LIN {X 0,Y 234.968,Z 259.216,A -85,B 0,C 180,E1 -19822.885,E2 -19822.885} C_VEL
LIN {X 0,Y 234.975,Z 259.214,A -85,B 0,C 180,E1 -19826.659,E2 -19826.659} C_VEL
LIN {X 0,Y 234.93,Z 259.221,A -85,B 0,C 180,E1 -19830.571,E2 -19830.571} C_VEL
LIN {X 0,Y 234.94,Z 259.221,A -85,B 0,C 180,E1 -19834.639,E2 -19834.639} C_VEL
LIN {X 0,Y 235.025,Z 259.387,A -85,B 0,C 180,E1 -19836.361,E2 -19836.361} C_VEL
LIN {X 0,Y 235.772,Z 263.846,A -85,B 0,C 180,E1 -19840.982,E2 -19840.982} C_VEL
LIN {X 0,Y 236.606,Z 268.443,A -85,B 0,C 180,E1 -19845.473,E2 -19845.473} C_VEL
LIN {X 0,Y 237.453,Z 272.706,A -85,B 0,C 180,E1 -19849.371,E2 -19849.371} C_VEL
LIN {X 0,Y 237.77,Z 275.178,A -85,B 0,C 180,E1 -19851.538,E2 -19851.538} C_VEL
LIN {X 0,Y 237.539,Z 276.271,A -85,B 0,C 180,E1 -19852.442,E2 -19852.442} C_VEL
LIN {X 0,Y 236.676,Z 277.419,A -85,B 0,C 180,E1 -19853.326,E2 -19853.326} C_VEL
LIN {X 0,Y 233.876,Z 279.774,A -85,B 0,C 180,E1 -19855.046,E2 -19855.046} C_VEL
LIN {X 0,Y 230.833,Z 282.181,A -85,B 0,C 180,E1 -19856.803,E2 -19856.803} C_VEL
LIN {X 0,Y 229.345,Z 283.979,A -85,B 0,C 180,E1 -19858.189,E2 -19858.189} C_VEL
LIN {X 0,Y 229.137,Z 284.57,A -85,B 0,C 180,E1 -19858.667,E2 -19858.667} C_VEL
LIN {X 0,Y 228.747,Z 286.319,A -85,B 0,C 180,E1 -19860.094,E2 -19860.094} C_VEL
LIN {X 0,Y 231.153,Z 300.125,A -85,B 0,C 180,E1 -19861.215,E2 -19861.215} C_VEL
LIN {X 0,Y 232.977,Z 313.771,A -85,B 0,C 180,E1 -19862.666,E2 -19862.666} C_VEL
LIN {X 0,Y 234.069,Z 325.973,A -85,B 0,C 180,E1 -19864.263,E2 -19864.263} C_VEL
LIN {X 0,Y 234.595,Z 337.731,A -85,B 0,C 180,E1 -19866.144,E2 -19866.144} C_VEL
LIN {X 0,Y 234.553,Z 342.841,A -85,B 0,C 180,E1 -19867.074,E2 -19867.074} C_VEL
LIN {X 0,Y 232.73,Z 351.383,A -85,B 0,C 180,E1 -19868.753,E2 -19868.753} C_VEL
LIN {X 0,Y 230.779,Z 360.913,A -85,B 0,C 180,E1 -19871.069,E2 -19871.069} C_VEL
LIN {X 0,Y 229.119,Z 368.99,A -85,B 0,C 180,E1 -19873.516,E2 -19873.516} C_VEL
LIN {X 0,Y 227.674,Z 375.926,A -85,B 0,C 180,E1 -19876.158,E2 -19876.158} C_VEL
LIN {X 0,Y 226.624,Z 382.296,A -85,B 0,C 180,E1 -19879.276,E2 -19879.276} C_VEL
LIN {X 0,Y 226.093,Z 386.448,A -85,B 0,C 180,E1 -19881.958,E2 -19881.958} C_VEL
LIN {X 0,Y 225.93,Z 389.517,A -85,B 0,C 180,E1 -19884.644,E2 -19884.644} C_VEL
LIN {X 0,Y 225.896,Z 391.02,A -85,B 0,C 180,E1 -19886.432,E2 -19886.432} C_VEL
LIN {X 0,Y 225.902,Z 392.054,A -85,B 0,C 180,E1 -19888.216,E2 -19888.216} C_VEL
LIN {X 0,Y 225.952,Z 392.675,A -85,B 0,C 180,E1 -19889.999,E2 -19889.999} C_VEL
LIN {X 0,Y 225.889,Z 392.888,A -85,B 0,C 180,E1 -19891.782,E2 -19891.782} C_VEL
LIN {X 0,Y 225.836,Z 392.705,A -85,B 0,C 180,E1 -19893.567,E2 -19893.567} C_VEL
LIN {X 0,Y 225.85,Z 392.091,A -85,B 0,C 180,E1 -19895.356,E2 -19895.356} C_VEL
LIN {X 0,Y 226.172,Z 389.669,A -85,B 0,C 180,E1 -19898.937,E2 -19898.937} C_VEL
LIN {X 0,Y 226.872,Z 386.782,A -85,B 0,C 180,E1 -19901.615,E2 -19901.615} C_VEL
LIN {X 0,Y 227.949,Z 382.909,A -85,B 0,C 180,E1 -19904.278,E2 -19904.278} C_VEL
LIN {X 0,Y 229.699,Z 377.964,A -85,B 0,C 180,E1 -19906.897,E2 -19906.897} C_VEL
LIN {X 0,Y 231.812,Z 371.807,A -85,B 0,C 180,E1 -19909.48,E2 -19909.48} C_VEL
LIN {X 0,Y 234.196,Z 364.248,A -85,B 0,C 180,E1 -19912.03,E2 -19912.03} C_VEL
LIN {X 0,Y 236.743,Z 356.653,A -85,B 0,C 180,E1 -19914.09,E2 -19914.09} C_VEL
LIN {X 0,Y 239.503,Z 347.574,A -85,B 0,C 180,E1 -19916.113,E2 -19916.113} C_VEL
LIN {X 0,Y 240.749,Z 336.486,A -85,B 0,C 180,E1 -19918.353,E2 -19918.353} C_VEL
LIN {X 0,Y 240.901,Z 325.735,A -85,B 0,C 180,E1 -19920.292,E2 -19920.292} C_VEL
LIN {X 0,Y 239.993,Z 315.116,A -85,B 0,C 180,E1 -19922.104,E2 -19922.104} C_VEL
LIN {X 0,Y 238.133,Z 304.29,A -85,B 0,C 180,E1 -19923.87,E2 -19923.87} C_VEL
LIN {X 0,Y 234.398,Z 291.005,A -85,B 0,C 180,E1 -19926.087,E2 -19926.087} C_VEL
LIN {X 0,Y 232.93,Z 286.928,A -85,B 0,C 180,E1 -19926.783,E2 -19926.783} C_VEL
LIN {X 0,Y 231.631,Z 283.737,A -85,B 0,C 180,E1 -19927.359,E2 -19927.359} C_VEL
LIN {X 0,Y 231.38,Z 282.361,A -85,B 0,C 180,E1 -19927.584,E2 -19927.584} C_VEL
LIN {X 0,Y 231.276,Z 279.496,A -85,B 0,C 180,E1 -19930.559,E2 -19930.559} C_VEL
LIN {X 0,Y 230.731,Z 276.118,A -85,B 0,C 180,E1 -19934.471,E2 -19934.471} C_VEL
LIN {X 0,Y 230.294,Z 273.504,A -85,B 0,C 180,E1 -19937.823,E2 -19937.823} C_VEL
LIN {X 0,Y 229.789,Z 270.45,A -85,B 0,C 180,E1 -19942.285,E2 -19942.285} C_VEL
LIN {X 0,Y 229.339,Z 268.039,A -85,B 0,C 180,E1 -19946.52,E2 -19946.52} C_VEL
LIN {X 0,Y 229.005,Z 266.125,A -85,B 0,C 180,E1 -19950.589,E2 -19950.589} C_VEL
LIN {X 0,Y 228.784,Z 264.663,A -85,B 0,C 180,E1 -19954.526,E2 -19954.526} C_VEL
LIN {X 0,Y 228.596,Z 263.623,A -85,B 0,C 180,E1 -19958.348,E2 -19958.348} C_VEL
LIN {X 0,Y 228.533,Z 262.899,A -85,B 0,C 180,E1 -19962.423,E2 -19962.423} C_VEL
LIN {X 0,Y 228.531,Z 262.566,A -85,B 0,C 180,E1 -19965.755,E2 -19965.755} C_VEL
LIN {X 0,Y 228.671,Z 262.482,A -85,B 0,C 180,E1 -19969.567,E2 -19969.567} C_VEL
LIN {X 0,Y 228.775,Z 262.67,A -85,B 0,C 180,E1 -19972.939,E2 -19972.939} C_VEL
LIN {X 0,Y 229.094,Z 263.408,A -85,B 0,C 180,E1 -19978.239,E2 -19978.239} C_VEL
LIN {X 0,Y 229.288,Z 263.758,A -85,B 0,C 180,E1 -19979.997,E2 -19979.997} C_VEL
LIN {X 0,Y 229.113,Z 265.292,A -85,B 0,C 180,E1 -19985.277,E2 -19985.277} C_VEL
LIN {X 0,Y 229.191,Z 266.612,A -85,B 0,C 180,E1 -19989.039,E2 -19989.039} C_VEL
LIN {X 0,Y 230.476,Z 269.741,A -85,B 0,C 180,E1 -19989.707,E2 -19989.707} C_VEL
LIN {X 0,Y 231.953,Z 271.819,A -85,B 0,C 180,E1 -19990.289,E2 -19990.289} C_VEL
LIN {X 0,Y 235.796,Z 279.227,A -85,B 0,C 180,E1 -19992.039,E2 -19992.039} C_VEL
LIN {X 0,Y 239.845,Z 288.945,A -85,B 0,C 180,E1 -19994.164,E2 -19994.164} C_VEL
LIN {X 0,Y 242.982,Z 299.405,A -85,B 0,C 180,E1 -19996.377,E2 -19996.377} C_VEL
LIN {X 0,Y 244.71,Z 309.094,A -85,B 0,C 180,E1 -19998.413,E2 -19998.413} C_VEL
LIN {X 0,Y 245.106,Z 313.998,A -85,B 0,C 180,E1 -19999.467,E2 -19999.467} C_VEL
LIN {X 0,Y 242.135,Z 324.686,A -85,B 0,C 180,E1 -20001.409,E2 -20001.409} C_VEL
LIN {X 0,Y 239.125,Z 334.171,A -85,B 0,C 180,E1 -20003.601,E2 -20003.601} C_VEL
LIN {X 0,Y 236.313,Z 342.387,A -85,B 0,C 180,E1 -20005.999,E2 -20005.999} C_VEL
LIN {X 0,Y 233.458,Z 349.872,A -85,B 0,C 180,E1 -20008.79,E2 -20008.79} C_VEL
LIN {X 0,Y 231.136,Z 355.679,A -85,B 0,C 180,E1 -20011.641,E2 -20011.641} C_VEL
LIN {X 0,Y 229.446,Z 359.674,A -85,B 0,C 180,E1 -20014.208,E2 -20014.208} C_VEL
LIN {X 0,Y 228.148,Z 362.637,A -85,B 0,C 180,E1 -20016.784,E2 -20016.784} C_VEL
LIN {X 0,Y 227.137,Z 364.655,A -85,B 0,C 180,E1 -20019.329,E2 -20019.329} C_VEL
LIN {X 0,Y 226.411,Z 365.821,A -85,B 0,C 180,E1 -20021.844,E2 -20021.844} C_VEL
LIN {X 0,Y 225.954,Z 366.155,A -85,B 0,C 180,E1 -20024.327,E2 -20024.327} C_VEL
LIN {X 0,Y 225.751,Z 365.739,A -85,B 0,C 180,E1 -20026.774,E2 -20026.774} C_VEL
LIN {X 0,Y 225.78,Z 364.618,A -85,B 0,C 180,E1 -20029.182,E2 -20029.182} C_VEL
LIN {X 0,Y 226.089,Z 362.754,A -85,B 0,C 180,E1 -20031.561,E2 -20031.561} C_VEL
LIN {X 0,Y 226.821,Z 358.635,A -85,B 0,C 180,E1 -20035.027,E2 -20035.027} C_VEL
LIN {X 0,Y 227.584,Z 354.595,A -85,B 0,C 180,E1 -20037.5,E2 -20037.5} C_VEL
LIN {X 0,Y 228.855,Z 348.086,A -85,B 0,C 180,E1 -20040.572,E2 -20040.572} C_VEL
LIN {X 0,Y 230.47,Z 340.722,A -85,B 0,C 180,E1 -20043.271,E2 -20043.271} C_VEL
LIN {X 0,Y 232.279,Z 331.67,A -85,B 0,C 180,E1 -20045.893,E2 -20045.893} C_VEL
LIN {X 0,Y 234.23,Z 322.215,A -85,B 0,C 180,E1 -20048.082,E2 -20048.082} C_VEL
LIN {X 0,Y 236.047,Z 312.051,A -85,B 0,C 180,E1 -20049.978,E2 -20049.978} C_VEL
LIN {X 0,Y 237.456,Z 303.625,A -85,B 0,C 180,E1 -20051.27,E2 -20051.27} C_VEL
LIN {X 0,Y 235.73,Z 293.055,A -85,B 0,C 180,E1 -20052.901,E2 -20052.901} C_VEL
LIN {X 0,Y 233.046,Z 281.209,A -85,B 0,C 180,E1 -20054.477,E2 -20054.477} C_VEL
LIN {X 0,Y 229.531,Z 268.807,A -85,B 0,C 180,E1 -20055.879,E2 -20055.879} C_VEL
LIN {X 0,Y 227.267,Z 261.563,A -85,B 0,C 180,E1 -20056.59,E2 -20056.59} C_VEL
LIN {X 0,Y 227.547,Z 260.142,A -85,B 0,C 180,E1 -20059.322,E2 -20059.322} C_VEL
LIN {X 0,Y 228.133,Z 260.069,A -85,B 0,C 180,E1 -20062.923,E2 -20062.923} C_VEL
LIN {X 0,Y 228.542,Z 260.018,A -85,B 0,C 180,E1 -20068.239,E2 -20068.239} C_VEL
LIN {X 0,Y 228.542,Z 260.016,A -85,B 0,C 180,E1 -20071.763,E2 -20071.763} C_VEL
LIN {X 0,Y 228.342,Z 260.04,A -85,B 0,C 180,E1 -20077.073,E2 -20077.073} C_VEL
LIN {X 0,Y 228.15,Z 260.066,A -85,B 0,C 180,E1 -20080.652,E2 -20080.652} C_VEL
LIN {X 0,Y 228.053,Z 260.079,A -85,B 0,C 180,E1 -20086.103,E2 -20086.103} C_VEL
LIN {X 0,Y 227.959,Z 260.088,A -85,B 0,C 180,E1 -20089.825,E2 -20089.825} C_VEL
LIN {X 0,Y 227.929,Z 260.094,A -85,B 0,C 180,E1 -20093.632,E2 -20093.632} C_VEL
LIN {X 0,Y 227.876,Z 260.096,A -85,B 0,C 180,E1 -20097.557,E2 -20097.557} C_VEL
LIN {X 0,Y 227.863,Z 260.101,A -85,B 0,C 180,E1 -20101.624,E2 -20101.624} C_VEL
LIN {X 0,Y 227.892,Z 260.09,A -85,B 0,C 180,E1 -20105.871,E2 -20105.871} C_VEL
LIN {X 0,Y 227.896,Z 260.097,A -85,B 0,C 180,E1 -20110.363,E2 -20110.363} C_VEL
LIN {X 0,Y 227.913,Z 260.091,A -85,B 0,C 180,E1 -20114.832,E2 -20114.832} C_VEL
LIN {X 0,Y 227.928,Z 260.081,A -85,B 0,C 180,E1 -20117.735,E2 -20117.735} C_VEL
LIN {X 0,Y 227.875,Z 260.098,A -85,B 0,C 180,E1 -20121.92,E2 -20121.92} C_VEL
LIN {X 0,Y 227.886,Z 260.096,A -85,B 0,C 180,E1 -20126.376,E2 -20126.376} C_VEL
LIN {X 0,Y 227.915,Z 260.085,A -85,B 0,C 180,E1 -20130.441,E2 -20130.441} C_VEL
LIN {X 0,Y 227.926,Z 260.093,A -85,B 0,C 180,E1 -20134.429,E2 -20134.429} C_VEL
LIN {X 0,Y 227.961,Z 260.087,A -85,B 0,C 180,E1 -20138.29,E2 -20138.29} C_VEL
LIN {X 0,Y 228.035,Z 260.067,A -85,B 0,C 180,E1 -20142.829,E2 -20142.829} C_VEL
LIN {X 0,Y 228.073,Z 260.073,A -85,B 0,C 180,E1 -20147.546,E2 -20147.546} C_VEL
LIN {X 0,Y 228.265,Z 260.049,A -85,B 0,C 180,E1 -20151.148,E2 -20151.148} C_VEL
LIN {X 0,Y 228.32,Z 260.038,A -85,B 0,C 180,E1 -20152.931,E2 -20152.931} C_VEL
LIN {X 0,Y 228.557,Z 260.012,A -85,B 0,C 180,E1 -20158.241,E2 -20158.241} C_VEL
LIN {X 0,Y 228.556,Z 260.017,A -85,B 0,C 180,E1 -20161.765,E2 -20161.765} C_VEL
LIN {X 0,Y 228.315,Z 260.035,A -85,B 0,C 180,E1 -20167.076,E2 -20167.076} C_VEL
LIN {X 0,Y 228.15,Z 260.063,A -85,B 0,C 180,E1 -20170.654,E2 -20170.654} C_VEL
LIN {X 0,Y 228.068,Z 260.072,A -85,B 0,C 180,E1 -20174.275,E2 -20174.275} C_VEL
LIN {X 0,Y 228.01,Z 260.081,A -85,B 0,C 180,E1 -20177.956,E2 -20177.956} C_VEL
LIN {X 0,Y 227.938,Z 260.091,A -85,B 0,C 180,E1 -20182.331,E2 -20182.331} C_VEL
LIN {X 0,Y 227.95,Z 260.09,A -85,B 0,C 180,E1 -20186.604,E2 -20186.604} C_VEL
LIN {X 0,Y 227.905,Z 260.095,A -85,B 0,C 180,E1 -20190.293,E2 -20190.293} C_VEL
LIN {X 0,Y 227.941,Z 260.093,A -85,B 0,C 180,E1 -20195.66,E2 -20195.66} C_VEL
LIN {X 0,Y 228.549,Z 263.853,A -85,B 0,C 180,E1 -20199.756,E2 -20199.756} C_VEL
LIN {X 0,Y 229.234,Z 267.624,A -85,B 0,C 180,E1 -20203.618,E2 -20203.618} C_VEL
LIN {X 0,Y 230.1,Z 271.927,A -85,B 0,C 180,E1 -20207.781,E2 -20207.781} C_VEL
LIN {X 0,Y 230.71,Z 275.958,A -85,B 0,C 180,E1 -20211.467,E2 -20211.467} C_VEL
LIN {X 0,Y 230.34,Z 279.576,A -85,B 0,C 180,E1 -20214.568,E2 -20214.568} C_VEL
LIN {X 0,Y 229.137,Z 284.57,A -85,B 0,C 180,E1 -20218.667,E2 -20218.667} C_VEL
LIN {X 0,Y 228.886,Z 286.269,A -85,B 0,C 180,E1 -20219.369,E2 -20219.369} C_VEL
LIN {X 0,Y 228.442,Z 289.896,A -85,B 0,C 180,E1 -20220.027,E2 -20220.027} C_VEL
LIN {X 0,Y 227.746,Z 295.552,A -85,B 0,C 180,E1 -20220.531,E2 -20220.531} C_VEL
LIN {X 0,Y 226.19,Z 306.821,A -85,B 0,C 180,E1 -20221.327,E2 -20221.327} C_VEL
LIN {X 0,Y 226.038,Z 313.153,A -85,B 0,C 180,E1 -20221.971,E2 -20221.971} C_VEL
LIN {X 0,Y 227.096,Z 325.04,A -85,B 0,C 180,E1 -20223.563,E2 -20223.563} C_VEL
LIN {X 0,Y 227.636,Z 336.145,A -85,B 0,C 180,E1 -20225.367,E2 -20225.367} C_VEL
LIN {X 0,Y 227.471,Z 343.759,A -85,B 0,C 180,E1 -20226.8,E2 -20226.8} C_VEL
LIN {X 0,Y 225.655,Z 352.086,A -85,B 0,C 180,E1 -20228.533,E2 -20228.533} C_VEL
LIN {X 0,Y 223.699,Z 361.369,A -85,B 0,C 180,E1 -20230.906,E2 -20230.906} C_VEL
LIN {X 0,Y 222.002,Z 369.289,A -85,B 0,C 180,E1 -20233.445,E2 -20233.445} C_VEL
LIN {X 0,Y 220.535,Z 376.088,A -85,B 0,C 180,E1 -20236.171,E2 -20236.171} C_VEL
LIN {X 0,Y 219.619,Z 381.53,A -85,B 0,C 180,E1 -20238.929,E2 -20238.929} C_VEL
LIN {X 0,Y 219.055,Z 385.761,A -85,B 0,C 180,E1 -20241.698,E2 -20241.698} C_VEL
LIN {X 0,Y 218.895,Z 388.906,A -85,B 0,C 180,E1 -20244.472,E2 -20244.472} C_VEL
LIN {X 0,Y 218.818,Z 390.443,A -85,B 0,C 180,E1 -20246.316,E2 -20246.316} C_VEL
LIN {X 0,Y 218.834,Z 391.542,A -85,B 0,C 180,E1 -20248.159,E2 -20248.159} C_VEL
LIN {X 0,Y 218.88,Z 392.194,A -85,B 0,C 180,E1 -20249.999,E2 -20249.999} C_VEL
LIN {X 0,Y 218.819,Z 392.439,A -85,B 0,C 180,E1 -20251.84,E2 -20251.84} C_VEL
LIN {X 0,Y 218.774,Z 391.862,A -85,B 0,C 180,E1 -20255.192,E2 -20255.192} C_VEL
LIN {X 0,Y 218.862,Z 390.765,A -85,B 0,C 180,E1 -20257.379,E2 -20257.379} C_VEL
LIN {X 0,Y 219.595,Z 387.639,A -85,B 0,C 180,E1 -20261.07,E2 -20261.07} C_VEL
LIN {X 0,Y 220.583,Z 384.174,A -85,B 0,C 180,E1 -20263.824,E2 -20263.824} C_VEL
LIN {X 0,Y 222.242,Z 379.682,A -85,B 0,C 180,E1 -20266.534,E2 -20266.534} C_VEL
LIN {X 0,Y 224.7,Z 373.034,A -85,B 0,C 180,E1 -20269.646,E2 -20269.646} C_VEL
LIN {X 0,Y 227.17,Z 365.861,A -85,B 0,C 180,E1 -20272.269,E2 -20272.269} C_VEL
LIN {X 0,Y 230.312,Z 357.056,A -85,B 0,C 180,E1 -20274.807,E2 -20274.807} C_VEL
LIN {X 0,Y 232.709,Z 350.054,A -85,B 0,C 180,E1 -20276.452,E2 -20276.452} C_VEL
LIN {X 0,Y 234.258,Z 339.819,A -85,B 0,C 180,E1 -20278.685,E2 -20278.685} C_VEL
LIN {X 0,Y 234.848,Z 330.187,A -85,B 0,C 180,E1 -20280.579,E2 -20280.579} C_VEL
LIN {X 0,Y 234.313,Z 318.822,A -85,B 0,C 180,E1 -20282.675,E2 -20282.675} C_VEL
LIN {X 0,Y 232.75,Z 307.621,A -85,B 0,C 180,E1 -20284.644,E2 -20284.644} C_VEL
LIN {X 0,Y 229.499,Z 294.855,A -85,B 0,C 180,E1 -20286.943,E2 -20286.943} C_VEL
LIN {X 0,Y 227.903,Z 290.354,A -85,B 0,C 180,E1 -20287.808,E2 -20287.808} C_VEL
LIN {X 0,Y 226.657,Z 286.91,A -85,B 0,C 180,E1 -20288.466,E2 -20288.466} C_VEL
LIN {X 0,Y 224.857,Z 283.567,A -85,B 0,C 180,E1 -20289.282,E2 -20289.282} C_VEL
LIN {X 0,Y 224.416,Z 281.713,A -85,B 0,C 180,E1 -20289.576,E2 -20289.576} C_VEL
LIN {X 0,Y 223.899,Z 278.116,A -85,B 0,C 180,E1 -20293.781,E2 -20293.781} C_VEL
LIN {X 0,Y 223.242,Z 274.481,A -85,B 0,C 180,E1 -20298.612,E2 -20298.612} C_VEL
LIN {X 0,Y 222.783,Z 271.534,A -85,B 0,C 180,E1 -20303.171,E2 -20303.171} C_VEL
LIN {X 0,Y 222.31,Z 269.239,A -85,B 0,C 180,E1 -20307.488,E2 -20307.488} C_VEL
LIN {X 0,Y 222.047,Z 267.418,A -85,B 0,C 180,E1 -20311.653,E2 -20311.653} C_VEL
LIN {X 0,Y 221.826,Z 266.071,A -85,B 0,C 180,E1 -20315.675,E2 -20315.675} C_VEL
LIN {X 0,Y 221.662,Z 265.125,A -85,B 0,C 180,E1 -20319.585,E2 -20319.585} C_VEL
LIN {X 0,Y 221.643,Z 264.523,A -85,B 0,C 180,E1 -20323.416,E2 -20323.416} C_VEL
LIN {X 0,Y 221.619,Z 264.242,A -85,B 0,C 180,E1 -20327.171,E2 -20327.171} C_VEL
LIN {X 0,Y 221.845,Z 264.216,A -85,B 0,C 180,E1 -20330.883,E2 -20330.883} C_VEL
LIN {X 0,Y 221.832,Z 264.527,A -85,B 0,C 180,E1 -20334.543,E2 -20334.543} C_VEL
LIN {X 0,Y 222.176,Z 265.025,A -85,B 0,C 180,E1 -20338.184,E2 -20338.184} C_VEL
LIN {X 0,Y 222.363,Z 265.346,A -85,B 0,C 180,E1 -20339.997,E2 -20339.997} C_VEL
LIN {X 0,Y 222.164,Z 266.305,A -85,B 0,C 180,E1 -20343.624,E2 -20343.624} C_VEL
LIN {X 0,Y 222.271,Z 267.329,A -85,B 0,C 180,E1 -20346.978,E2 -20346.978} C_VEL
LIN {X 0,Y 223.527,Z 270.421,A -85,B 0,C 180,E1 -20347.676,E2 -20347.676} C_VEL
LIN {X 0,Y 225.456,Z 272.865,A -85,B 0,C 180,E1 -20348.512,E2 -20348.512} C_VEL
LIN {X 0,Y 227.344,Z 276.202,A -85,B 0,C 180,E1 -20349.441,E2 -20349.441} C_VEL
LIN {X 0,Y 231.257,Z 284.148,A -85,B 0,C 180,E1 -20351.45,E2 -20351.45} C_VEL
LIN {X 0,Y 235.059,Z 294.303,A -85,B 0,C 180,E1 -20353.836,E2 -20353.836} C_VEL
LIN {X 0,Y 237.429,Z 303.385,A -85,B 0,C 180,E1 -20355.888,E2 -20355.888} C_VEL
LIN {X 0,Y 238.808,Z 312.702,A -85,B 0,C 180,E1 -20357.996,E2 -20357.996} C_VEL
LIN {X 0,Y 239.049,Z 315.526,A -85,B 0,C 180,E1 -20358.653,E2 -20358.653} C_VEL
LIN {X 0,Y 236.225,Z 325.137,A -85,B 0,C 180,E1 -20360.458,E2 -20360.458} C_VEL
LIN {X 0,Y 233.007,Z 334.695,A -85,B 0,C 180,E1 -20362.722,E2 -20362.722} C_VEL
LIN {X 0,Y 229.837,Z 343.388,A -85,B 0,C 180,E1 -20365.343,E2 -20365.343} C_VEL
LIN {X 0,Y 227.401,Z 349.398,A -85,B 0,C 180,E1 -20367.615,E2 -20367.615} C_VEL
LIN {X 0,Y 225.313,Z 354.324,A -85,B 0,C 180,E1 -20369.935,E2 -20369.935} C_VEL
LIN {X 0,Y 223.53,Z 358.337,A -85,B 0,C 180,E1 -20372.306,E2 -20372.306} C_VEL
LIN {X 0,Y 222.035,Z 361.528,A -85,B 0,C 180,E1 -20374.728,E2 -20374.728} C_VEL
LIN {X 0,Y 220.827,Z 364.005,A -85,B 0,C 180,E1 -20377.286,E2 -20377.286} C_VEL
LIN {X 0,Y 219.863,Z 365.671,A -85,B 0,C 180,E1 -20379.902,E2 -20379.902} C_VEL
LIN {X 0,Y 219.183,Z 366.482,A -85,B 0,C 180,E1 -20382.484,E2 -20382.484} C_VEL
LIN {X 0,Y 218.774,Z 366.526,A -85,B 0,C 180,E1 -20385.031,E2 -20385.031} C_VEL
LIN {X 0,Y 218.664,Z 365.782,A -85,B 0,C 180,E1 -20387.661,E2 -20387.661} C_VEL
LIN {X 0,Y 218.819,Z 364.114,A -85,B 0,C 180,E1 -20390.422,E2 -20390.422} C_VEL
LIN {X 0,Y 219.503,Z 360.447,A -85,B 0,C 180,E1 -20394.044,E2 -20394.044} C_VEL
LIN {X 0,Y 220.338,Z 355.883,A -85,B 0,C 180,E1 -20397.165,E2 -20397.165} C_VEL
LIN {X 0,Y 221.506,Z 350.33,A -85,B 0,C 180,E1 -20400.02,E2 -20400.02} C_VEL
LIN {X 0,Y 223.152,Z 342.814,A -85,B 0,C 180,E1 -20403.018,E2 -20403.018} C_VEL
LIN {X 0,Y 224.873,Z 334.614,A -85,B 0,C 180,E1 -20405.616,E2 -20405.616} C_VEL
LIN {X 0,Y 226.786,Z 325.461,A -85,B 0,C 180,E1 -20407.931,E2 -20407.931} C_VEL
LIN {X 0,Y 228.794,Z 315.178,A -85,B 0,C 180,E1 -20410.019,E2 -20410.019} C_VEL
LIN {X 0,Y 230.676,Z 304.573,A -85,B 0,C 180,E1 -20411.746,E2 -20411.746} C_VEL
LIN {X 0,Y 228.759,Z 293.176,A -85,B 0,C 180,E1 -20413.58,E2 -20413.58} C_VEL
LIN {X 0,Y 226.135,Z 281.8,A -85,B 0,C 180,E1 -20415.145,E2 -20415.145} C_VEL
LIN {X 0,Y 222.615,Z 269.482,A -85,B 0,C 180,E1 -20416.595,E2 -20416.595} C_VEL
LIN {X 0,Y 220.286,Z 261.958,A -85,B 0,C 180,E1 -20417.389,E2 -20417.389} C_VEL
LIN {X 0,Y 220.423,Z 261.03,A -85,B 0,C 180,E1 -20418.972,E2 -20418.972} C_VEL
LIN {X 0,Y 220.843,Z 260.976,A -85,B 0,C 180,E1 -20420.845,E2 -20420.845} C_VEL
LIN {X 0,Y 221.053,Z 260.95,A -85,B 0,C 180,E1 -20422.695,E2 -20422.695} C_VEL
LIN {X 0,Y 221.499,Z 260.895,A -85,B 0,C 180,E1 -20428.183,E2 -20428.183} C_VEL
LIN {X 0,Y 221.5,Z 260.893,A -85,B 0,C 180,E1 -20431.819,E2 -20431.819} C_VEL
LIN {X 0,Y 221.277,Z 260.921,A -85,B 0,C 180,E1 -20437.3,E2 -20437.3} C_VEL
LIN {X 0,Y 221.099,Z 260.944,A -85,B 0,C 180,E1 -20440.996,E2 -20440.996} C_VEL
LIN {X 0,Y 221.013,Z 260.958,A -85,B 0,C 180,E1 -20446.631,E2 -20446.631} C_VEL
LIN {X 0,Y 220.914,Z 260.967,A -85,B 0,C 180,E1 -20450.485,E2 -20450.485} C_VEL
LIN {X 0,Y 220.872,Z 260.975,A -85,B 0,C 180,E1 -20454.435,E2 -20454.435} C_VEL
LIN {X 0,Y 220.827,Z 260.976,A -85,B 0,C 180,E1 -20458.516,E2 -20458.516} C_VEL
LIN {X 0,Y 220.814,Z 260.981,A -85,B 0,C 180,E1 -20462.757,E2 -20462.757} C_VEL
LIN {X 0,Y 220.829,Z 260.971,A -85,B 0,C 180,E1 -20467.291,E2 -20467.291} C_VEL
LIN {X 0,Y 220.866,Z 260.972,A -85,B 0,C 180,E1 -20471.931,E2 -20471.931} C_VEL
LIN {X 0,Y 220.868,Z 260.966,A -85,B 0,C 180,E1 -20475.575,E2 -20475.575} C_VEL
LIN {X 0,Y 220.855,Z 260.968,A -85,B 0,C 180,E1 -20479.795,E2 -20479.795} C_VEL
LIN {X 0,Y 220.834,Z 260.977,A -85,B 0,C 180,E1 -20482.799,E2 -20482.799} C_VEL
LIN {X 0,Y 220.821,Z 260.972,A -85,B 0,C 180,E1 -20487.249,E2 -20487.249} C_VEL
LIN {X 0,Y 220.833,Z 260.967,A -85,B 0,C 180,E1 -20491.49,E2 -20491.49} C_VEL
LIN {X 0,Y 220.865,Z 260.971,A -85,B 0,C 180,E1 -20495.569,E2 -20495.569} C_VEL
LIN {X 0,Y 220.892,Z 260.966,A -85,B 0,C 180,E1 -20499.517,E2 -20499.517} C_VEL
LIN {X 0,Y 221.017,Z 260.941,A -85,B 0,C 180,E1 -20503.374,E2 -20503.374} C_VEL
LIN {X 0,Y 221.013,Z 260.951,A -85,B 0,C 180,E1 -20507.142,E2 -20507.142} C_VEL
LIN {X 0,Y 221.203,Z 260.928,A -85,B 0,C 180,E1 -20510.863,E2 -20510.863} C_VEL
LIN {X 0,Y 221.138,Z 260.928,A -85,B 0,C 180,E1 -20514.532,E2 -20514.532} C_VEL
LIN {X 0,Y 221.515,Z 260.89,A -85,B 0,C 180,E1 -20518.185,E2 -20518.185} C_VEL
LIN {X 0,Y 221.514,Z 260.893,A -85,B 0,C 180,E1 -20521.821,E2 -20521.821} C_VEL
LIN {X 0,Y 221.252,Z 260.915,A -85,B 0,C 180,E1 -20527.303,E2 -20527.303} C_VEL
LIN {X 0,Y 221.072,Z 260.946,A -85,B 0,C 180,E1 -20530.999,E2 -20530.999} C_VEL
LIN {X 0,Y 221.023,Z 260.945,A -85,B 0,C 180,E1 -20536.632,E2 -20536.632} C_VEL
LIN {X 0,Y 220.9,Z 260.967,A -85,B 0,C 180,E1 -20540.488,E2 -20540.488} C_VEL
LIN {X 0,Y 220.875,Z 260.971,A -85,B 0,C 180,E1 -20544.437,E2 -20544.437} C_VEL
LIN {X 0,Y 220.835,Z 260.976,A -85,B 0,C 180,E1 -20548.517,E2 -20548.517} C_VEL
LIN {X 0,Y 220.825,Z 260.979,A -85,B 0,C 180,E1 -20552.758,E2 -20552.758} C_VEL
LIN {X 0,Y 220.877,Z 260.996,A -85,B 0,C 180,E1 -20555.223,E2 -20555.223} C_VEL
LIN {X 0,Y 221.254,Z 262.925,A -85,B 0,C 180,E1 -20557.427,E2 -20557.427} C_VEL
LIN {X 0,Y 221.897,Z 266.859,A -85,B 0,C 180,E1 -20561.695,E2 -20561.695} C_VEL
LIN {X 0,Y 222.786,Z 271.605,A -85,B 0,C 180,E1 -20566.519,E2 -20566.519} C_VEL
LIN {X 0,Y 223.477,Z 275.311,A -85,B 0,C 180,E1 -20570.071,E2 -20570.071} C_VEL
LIN {X 0,Y 223.647,Z 277.167,A -85,B 0,C 180,E1 -20571.781,E2 -20571.781} C_VEL
LIN {X 0,Y 223.513,Z 278.882,A -85,B 0,C 180,E1 -20573.313,E2 -20573.313} C_VEL
LIN {X 0,Y 222.349,Z 283.787,A -85,B 0,C 180,E1 -20577.497,E2 -20577.497} C_VEL
LIN {X 0,Y 221.883,Z 285.968,A -85,B 0,C 180,E1 -20579.337,E2 -20579.337} C_VEL
LIN {X 0,Y 224.328,Z 300.095,A -85,B 0,C 180,E1 -20580.542,E2 -20580.542} C_VEL
LIN {X 0,Y 226.038,Z 313.153,A -85,B 0,C 180,E1 -20581.971,E2 -20581.971} C_VEL
LIN {X 0,Y 225.877,Z 318.574,A -85,B 0,C 180,E1 -20582.594,E2 -20582.594} C_VEL
LIN {X 0,Y 223.763,Z 327.332,A -85,B 0,C 180,E1 -20583.633,E2 -20583.633} C_VEL
LIN {X 0,Y 221.358,Z 335.781,A -85,B 0,C 180,E1 -20584.842,E2 -20584.842} C_VEL
LIN {X 0,Y 220.763,Z 340.626,A -85,B 0,C 180,E1 -20585.721,E2 -20585.721} C_VEL
LIN {X 0,Y 220.379,Z 344.579,A -85,B 0,C 180,E1 -20586.506,E2 -20586.506} C_VEL
LIN {X 0,Y 218.232,Z 354.538,A -85,B 0,C 180,E1 -20588.758,E2 -20588.758} C_VEL
LIN {X 0,Y 216.456,Z 362.736,A -85,B 0,C 180,E1 -20591.053,E2 -20591.053} C_VEL
LIN {X 0,Y 214.634,Z 370.768,A -85,B 0,C 180,E1 -20593.839,E2 -20593.839} C_VEL
LIN {X 0,Y 213.19,Z 377.204,A -85,B 0,C 180,E1 -20596.657,E2 -20596.657} C_VEL
LIN {X 0,Y 212.38,Z 382.317,A -85,B 0,C 180,E1 -20599.513,E2 -20599.513} C_VEL
LIN {X 0,Y 211.879,Z 386.252,A -85,B 0,C 180,E1 -20602.375,E2 -20602.375} C_VEL
LIN {X 0,Y 211.801,Z 388.524,A -85,B 0,C 180,E1 -20604.565,E2 -20604.565} C_VEL
LIN {X 0,Y 211.767,Z 391.002,A -85,B 0,C 180,E1 -20608.097,E2 -20608.097} C_VEL
LIN {X 0,Y 211.81,Z 391.706,A -85,B 0,C 180,E1 -20609.999,E2 -20609.999} C_VEL
LIN {X 0,Y 211.75,Z 391.988,A -85,B 0,C 180,E1 -20611.901,E2 -20611.901} C_VEL
LIN {X 0,Y 211.692,Z 391.56,A -85,B 0,C 180,E1 -20615.116,E2 -20615.116} C_VEL
LIN {X 0,Y 211.795,Z 390.459,A -85,B 0,C 180,E1 -20617.626,E2 -20617.626} C_VEL
LIN {X 0,Y 212.579,Z 387.408,A -85,B 0,C 180,E1 -20621.44,E2 -20621.44} C_VEL
LIN {X 0,Y 213.673,Z 384.042,A -85,B 0,C 180,E1 -20624.28,E2 -20624.28} C_VEL
LIN {X 0,Y 215.433,Z 379.663,A -85,B 0,C 180,E1 -20627.073,E2 -20627.073} C_VEL
LIN {X 0,Y 217.583,Z 374.159,A -85,B 0,C 180,E1 -20629.824,E2 -20629.824} C_VEL
LIN {X 0,Y 220.148,Z 367.371,A -85,B 0,C 180,E1 -20632.524,E2 -20632.524} C_VEL
LIN {X 0,Y 223.297,Z 359.059,A -85,B 0,C 180,E1 -20635.143,E2 -20635.143} C_VEL
LIN {X 0,Y 226.353,Z 350.665,A -85,B 0,C 180,E1 -20637.255,E2 -20637.255} C_VEL
LIN {X 0,Y 228.08,Z 340.743,A -85,B 0,C 180,E1 -20639.538,E2 -20639.538} C_VEL
LIN {X 0,Y 228.786,Z 331.404,A -85,B 0,C 180,E1 -20641.48,E2 -20641.48} C_VEL
LIN {X 0,Y 228.371,Z 319.541,A -85,B 0,C 180,E1 -20643.804,E2 -20643.804} C_VEL
LIN {X 0,Y 226.908,Z 308.652,A -85,B 0,C 180,E1 -20645.878,E2 -20645.878} C_VEL
LIN {X 0,Y 223.933,Z 296.118,A -85,B 0,C 180,E1 -20648.312,E2 -20648.312} C_VEL
LIN {X 0,Y 222.113,Z 291.312,A -85,B 0,C 180,E1 -20649.379,E2 -20649.379} C_VEL
LIN {X 0,Y 220.479,Z 287.639,A -85,B 0,C 180,E1 -20650.258,E2 -20650.258} C_VEL
LIN {X 0,Y 219.61,Z 286.184,A -85,B 0,C 180,E1 -20650.672,E2 -20650.672} C_VEL
LIN {X 0,Y 217.643,Z 282.698,A -85,B 0,C 180,E1 -20651.675,E2 -20651.675} C_VEL
LIN {X 0,Y 217.155,Z 280.93,A -85,B 0,C 180,E1 -20652.041,E2 -20652.041} C_VEL
LIN {X 0,Y 216.636,Z 278.198,A -85,B 0,C 180,E1 -20655.536,E2 -20655.536} C_VEL
LIN {X 0,Y 216.221,Z 275.45,A -85,B 0,C 180,E1 -20659.449,E2 -20659.449} C_VEL
LIN {X 0,Y 215.749,Z 272.652,A -85,B 0,C 180,E1 -20664.099,E2 -20664.099} C_VEL
LIN {X 0,Y 215.391,Z 270.436,A -85,B 0,C 180,E1 -20668.526,E2 -20668.526} C_VEL
LIN {X 0,Y 215.106,Z 268.732,A -85,B 0,C 180,E1 -20672.777,E2 -20672.777} C_VEL
LIN {X 0,Y 214.913,Z 267.482,A -85,B 0,C 180,E1 -20676.892,E2 -20676.892} C_VEL
LIN {X 0,Y 214.774,Z 266.51,A -85,B 0,C 180,E1 -20681.611,E2 -20681.611} C_VEL
LIN {X 0,Y 214.75,Z 266.124,A -85,B 0,C 180,E1 -20684.819,E2 -20684.819} C_VEL
LIN {X 0,Y 214.949,Z 265.918,A -85,B 0,C 180,E1 -20690.588,E2 -20690.588} C_VEL
LIN {X 0,Y 214.951,Z 266.188,A -85,B 0,C 180,E1 -20694.368,E2 -20694.368} C_VEL
LIN {X 0,Y 215.263,Z 266.652,A -85,B 0,C 180,E1 -20698.126,E2 -20698.126} C_VEL
LIN {X 0,Y 215.464,Z 266.952,A -85,B 0,C 180,E1 -20699.997,E2 -20699.997} C_VEL
LIN {X 0,Y 215.284,Z 268.304,A -85,B 0,C 180,E1 -20704.561,E2 -20704.561} C_VEL
LIN {X 0,Y 216.369,Z 270.889,A -85,B 0,C 180,E1 -20705.238,E2 -20705.238} C_VEL
LIN {X 0,Y 218.727,Z 273.665,A -85,B 0,C 180,E1 -20706.397,E2 -20706.397} C_VEL
LIN {X 0,Y 220.5,Z 276.89,A -85,B 0,C 180,E1 -20707.379,E2 -20707.379} C_VEL
LIN {X 0,Y 221.503,Z 278.267,A -85,B 0,C 180,E1 -20707.868,E2 -20707.868} C_VEL
LIN {X 0,Y 226.408,Z 288.487,A -85,B 0,C 180,E1 -20710.731,E2 -20710.731} C_VEL
LIN {X 0,Y 229.337,Z 296.745,A -85,B 0,C 180,E1 -20712.834,E2 -20712.834} C_VEL
LIN {X 0,Y 231.579,Z 305.929,A -85,B 0,C 180,E1 -20715.064,E2 -20715.064} C_VEL
LIN {X 0,Y 232.713,Z 314.419,A -85,B 0,C 180,E1 -20717.121,E2 -20717.121} C_VEL
LIN {X 0,Y 232.766,Z 317.983,A -85,B 0,C 180,E1 -20717.971,E2 -20717.971} C_VEL
LIN {X 0,Y 229.348,Z 328.691,A -85,B 0,C 180,E1 -20720.149,E2 -20720.149} C_VEL
LIN {X 0,Y 226.163,Z 337.372,A -85,B 0,C 180,E1 -20722.371,E2 -20722.371} C_VEL
LIN {X 0,Y 223.309,Z 344.619,A -85,B 0,C 180,E1 -20724.715,E2 -20724.715} C_VEL
LIN {X 0,Y 220.819,Z 350.343,A -85,B 0,C 180,E1 -20726.984,E2 -20726.984} C_VEL
LIN {X 0,Y 217.857,Z 356.813,A -85,B 0,C 180,E1 -20730.331,E2 -20730.331} C_VEL
LIN {X 0,Y 215.545,Z 361.513,A -85,B 0,C 180,E1 -20733.658,E2 -20733.658} C_VEL
LIN {X 0,Y 214.221,Z 364.019,A -85,B 0,C 180,E1 -20736.19,E2 -20736.19} C_VEL
LIN {X 0,Y 213.128,Z 365.787,A -85,B 0,C 180,E1 -20738.79,E2 -20738.79} C_VEL
LIN {X 0,Y 212.323,Z 366.808,A -85,B 0,C 180,E1 -20741.448,E2 -20741.448} C_VEL
LIN {X 0,Y 211.781,Z 367.054,A -85,B 0,C 180,E1 -20744.173,E2 -20744.173} C_VEL
LIN {X 0,Y 211.565,Z 366.439,A -85,B 0,C 180,E1 -20746.949,E2 -20746.949} C_VEL
LIN {X 0,Y 211.651,Z 364.927,A -85,B 0,C 180,E1 -20749.788,E2 -20749.788} C_VEL
LIN {X 0,Y 212.251,Z 361.648,A -85,B 0,C 180,E1 -20753.417,E2 -20753.417} C_VEL
LIN {X 0,Y 212.83,Z 358.535,A -85,B 0,C 180,E1 -20755.851,E2 -20755.851} C_VEL
LIN {X 0,Y 213.806,Z 353.805,A -85,B 0,C 180,E1 -20758.713,E2 -20758.713} C_VEL
LIN {X 0,Y 215.275,Z 347.156,A -85,B 0,C 180,E1 -20761.81,E2 -20761.81} C_VEL
LIN {X 0,Y 216.923,Z 339.75,A -85,B 0,C 180,E1 -20764.538,E2 -20764.538} C_VEL
LIN {X 0,Y 218.827,Z 331.157,A -85,B 0,C 180,E1 -20767.083,E2 -20767.083} C_VEL
LIN {X 0,Y 221.021,Z 320.731,A -85,B 0,C 180,E1 -20769.527,E2 -20769.527} C_VEL
LIN {X 0,Y 223.274,Z 309.248,A -85,B 0,C 180,E1 -20771.654,E2 -20771.654} C_VEL
LIN {X 0,Y 223.85,Z 305.239,A -85,B 0,C 180,E1 -20772.29,E2 -20772.29} C_VEL
LIN {X 0,Y 221.934,Z 294.164,A -85,B 0,C 180,E1 -20774.151,E2 -20774.151} C_VEL
LIN {X 0,Y 219.228,Z 282.313,A -85,B 0,C 180,E1 -20775.852,E2 -20775.852} C_VEL
LIN {X 0,Y 215.583,Z 269.746,A -85,B 0,C 180,E1 -20777.408,E2 -20777.408} C_VEL
LIN {X 0,Y 213.3,Z 262.4,A -85,B 0,C 180,E1 -20778.177,E2 -20778.177} C_VEL
LIN {X 0,Y 213.705,Z 261.865,A -85,B 0,C 180,E1 -20780.584,E2 -20780.584} C_VEL
LIN {X 0,Y 213.977,Z 261.832,A -85,B 0,C 180,E1 -20782.452,E2 -20782.452} C_VEL
LIN {X 0,Y 214.431,Z 261.776,A -85,B 0,C 180,E1 -20788.123,E2 -20788.123} C_VEL
LIN {X 0,Y 214.541,Z 261.762,A -85,B 0,C 180,E1 -20790.001,E2 -20790.001} C_VEL
LIN {X 0,Y 214.433,Z 261.773,A -85,B 0,C 180,E1 -20791.879,E2 -20791.879} C_VEL
LIN {X 0,Y 214.215,Z 261.801,A -85,B 0,C 180,E1 -20797.542,E2 -20797.542} C_VEL
LIN {X 0,Y 214.032,Z 261.821,A -85,B 0,C 180,E1 -20801.364,E2 -20801.364} C_VEL
LIN {X 0,Y 213.926,Z 261.841,A -85,B 0,C 180,E1 -20805.238,E2 -20805.238} C_VEL
LIN {X 0,Y 213.873,Z 261.843,A -85,B 0,C 180,E1 -20809.185,E2 -20809.185} C_VEL
LIN {X 0,Y 213.852,Z 261.85,A -85,B 0,C 180,E1 -20813.227,E2 -20813.227} C_VEL
LIN {X 0,Y 213.818,Z 261.847,A -85,B 0,C 180,E1 -20817.452,E2 -20817.452} C_VEL
LIN {X 0,Y 213.77,Z 261.857,A -85,B 0,C 180,E1 -20821.738,E2 -20821.738} C_VEL
LIN {X 0,Y 213.745,Z 261.852,A -85,B 0,C 180,E1 -20826.289,E2 -20826.289} C_VEL
LIN {X 0,Y 213.817,Z 261.851,A -85,B 0,C 180,E1 -20831.102,E2 -20831.102} C_VEL
LIN {X 0,Y 213.829,Z 261.847,A -85,B 0,C 180,E1 -20833.696,E2 -20833.696} C_VEL
LIN {X 0,Y 213.834,Z 261.84,A -85,B 0,C 180,E1 -20836.359,E2 -20836.359} C_VEL
LIN {X 0,Y 213.818,Z 261.844,A -85,B 0,C 180,E1 -20839.113,E2 -20839.113} C_VEL
LIN {X 0,Y 213.752,Z 261.858,A -85,B 0,C 180,E1 -20843.718,E2 -20843.718} C_VEL
LIN {X 0,Y 213.792,Z 261.842,A -85,B 0,C 180,E1 -20848.728,E2 -20848.728} C_VEL
LIN {X 0,Y 213.823,Z 261.846,A -85,B 0,C 180,E1 -20852.607,E2 -20852.607} C_VEL
LIN {X 0,Y 213.851,Z 261.845,A -85,B 0,C 180,E1 -20856.956,E2 -20856.956} C_VEL
LIN {X 0,Y 213.944,Z 261.821,A -85,B 0,C 180,E1 -20862.807,E2 -20862.807} C_VEL
LIN {X 0,Y 213.954,Z 261.831,A -85,B 0,C 180,E1 -20866.71,E2 -20866.71} C_VEL
LIN {X 0,Y 214.141,Z 261.808,A -85,B 0,C 180,E1 -20870.559,E2 -20870.559} C_VEL
LIN {X 0,Y 214.099,Z 261.804,A -85,B 0,C 180,E1 -20874.352,E2 -20874.352} C_VEL
LIN {X 0,Y 214.448,Z 261.77,A -85,B 0,C 180,E1 -20878.125,E2 -20878.125} C_VEL
LIN {X 0,Y 214.554,Z 261.76,A -85,B 0,C 180,E1 -20880.003,E2 -20880.003} C_VEL
LIN {X 0,Y 214.447,Z 261.773,A -85,B 0,C 180,E1 -20881.881,E2 -20881.881} C_VEL
LIN {X 0,Y 214.192,Z 261.795,A -85,B 0,C 180,E1 -20887.545,E2 -20887.545} C_VEL
LIN {X 0,Y 214.004,Z 261.828,A -85,B 0,C 180,E1 -20891.367,E2 -20891.367} C_VEL
LIN {X 0,Y 213.939,Z 261.832,A -85,B 0,C 180,E1 -20895.24,E2 -20895.24} C_VEL
LIN {X 0,Y 213.847,Z 261.846,A -85,B 0,C 180,E1 -20899.19,E2 -20899.19} C_VEL
LIN {X 0,Y 213.855,Z 261.848,A -85,B 0,C 180,E1 -20903.229,E2 -20903.229} C_VEL
LIN {X 0,Y 213.837,Z 261.85,A -85,B 0,C 180,E1 -20907.452,E2 -20907.452} C_VEL
LIN {X 0,Y 213.776,Z 261.857,A -85,B 0,C 180,E1 -20911.739,E2 -20911.739} C_VEL
LIN {X 0,Y 213.83,Z 261.9,A -85,B 0,C 180,E1 -20914.745,E2 -20914.745} C_VEL
LIN {X 0,Y 214.553,Z 266.176,A -85,B 0,C 180,E1 -20919.702,E2 -20919.702} C_VEL
LIN {X 0,Y 215.281,Z 270.243,A -85,B 0,C 180,E1 -20924.092,E2 -20924.092} C_VEL
LIN {X 0,Y 216.159,Z 274.484,A -85,B 0,C 180,E1 -20928.404,E2 -20928.404} C_VEL
LIN {X 0,Y 216.559,Z 278.132,A -85,B 0,C 180,E1 -20931.93,E2 -20931.93} C_VEL
LIN {X 0,Y 216.144,Z 280.841,A -85,B 0,C 180,E1 -20934.383,E2 -20934.383} C_VEL
LIN {X 0,Y 214.99,Z 285.553,A -85,B 0,C 180,E1 -20938.526,E2 -20938.526} C_VEL
LIN {X 0,Y 217.464,Z 299.872,A -85,B 0,C 180,E1 -20939.805,E2 -20939.805} C_VEL
LIN {X 0,Y 219.251,Z 313.785,A -85,B 0,C 180,E1 -20941.404,E2 -20941.404} C_VEL
LIN {X 0,Y 220.248,Z 325.451,A -85,B 0,C 180,E1 -20943.05,E2 -20943.05} C_VEL
LIN {X 0,Y 220.734,Z 337.109,A -85,B 0,C 180,E1 -20945.046,E2 -20945.046} C_VEL
LIN {X 0,Y 220.763,Z 340.626,A -85,B 0,C 180,E1 -20945.721,E2 -20945.721} C_VEL
LIN {X 0,Y 219.896,Z 343.77,A -85,B 0,C 180,E1 -20946.305,E2 -20946.305} C_VEL
LIN {X 0,Y 217.9,Z 346.692,A -85,B 0,C 180,E1 -20946.814,E2 -20946.814} C_VEL
LIN {X 0,Y 212.337,Z 352.998,A -85,B 0,C 180,E1 -20948.027,E2 -20948.027} C_VEL
LIN {X 0,Y 210.992,Z 355.788,A -85,B 0,C 180,E1 -20948.726,E2 -20948.726} C_VEL
LIN {X 0,Y 209.01,Z 364.532,A -85,B 0,C 180,E1 -20951.37,E2 -20951.37} C_VEL
LIN {X 0,Y 207.261,Z 372.093,A -85,B 0,C 180,E1 -20954.259,E2 -20954.259} C_VEL
LIN {X 0,Y 205.902,Z 378.161,A -85,B 0,C 180,E1 -20957.181,E2 -20957.181} C_VEL
LIN {X 0,Y 205.147,Z 382.969,A -85,B 0,C 180,E1 -20960.136,E2 -20960.136} C_VEL
LIN {X 0,Y 204.749,Z 386.627,A -85,B 0,C 180,E1 -20963.099,E2 -20963.099} C_VEL
LIN {X 0,Y 204.675,Z 389.239,A -85,B 0,C 180,E1 -20966.061,E2 -20966.061} C_VEL
LIN {X 0,Y 204.702,Z 390.439,A -85,B 0,C 180,E1 -20968.031,E2 -20968.031} C_VEL
LIN {X 0,Y 204.741,Z 391.216,A -85,B 0,C 180,E1 -20969.999,E2 -20969.999} C_VEL
LIN {X 0,Y 204.68,Z 391.537,A -85,B 0,C 180,E1 -20971.967,E2 -20971.967} C_VEL
LIN {X 0,Y 204.586,Z 390.993,A -85,B 0,C 180,E1 -20975.914,E2 -20975.914} C_VEL
LIN {X 0,Y 204.721,Z 390.147,A -85,B 0,C 180,E1 -20977.892,E2 -20977.892} C_VEL
LIN {X 0,Y 205.068,Z 388.879,A -85,B 0,C 180,E1 -20979.866,E2 -20979.866} C_VEL
LIN {X 0,Y 206.279,Z 385.132,A -85,B 0,C 180,E1 -20983.796,E2 -20983.796} C_VEL
LIN {X 0,Y 207.96,Z 381.191,A -85,B 0,C 180,E1 -20986.693,E2 -20986.693} C_VEL
LIN {X 0,Y 210.045,Z 376.177,A -85,B 0,C 180,E1 -20989.547,E2 -20989.547} C_VEL
LIN {X 0,Y 212.824,Z 369.641,A -85,B 0,C 180,E1 -20992.473,E2 -20992.473} C_VEL
LIN {X 0,Y 215.738,Z 362.408,A -85,B 0,C 180,E1 -20995.054,E2 -20995.054} C_VEL
LIN {X 0,Y 219.497,Z 353.038,A -85,B 0,C 180,E1 -20997.662,E2 -20997.662} C_VEL
LIN {X 0,Y 221.395,Z 344.717,A -85,B 0,C 180,E1 -20999.735,E2 -20999.735} C_VEL
LIN {X 0,Y 222.612,Z 334.953,A -85,B 0,C 180,E1 -21001.93,E2 -21001.93} C_VEL
LIN {X 0,Y 222.719,Z 324.229,A -85,B 0,C 180,E1 -21004.215,E2 -21004.215} C_VEL
LIN {X 0,Y 221.754,Z 313.166,A -85,B 0,C 180,E1 -21006.464,E2 -21006.464} C_VEL
LIN {X 0,Y 219.653,Z 302.214,A -85,B 0,C 180,E1 -21008.757,E2 -21008.757} C_VEL
LIN {X 0,Y 217.631,Z 295.876,A -85,B 0,C 180,E1 -21010.229,E2 -21010.229} C_VEL
LIN {X 0,Y 215.729,Z 291.477,A -85,B 0,C 180,E1 -21011.411,E2 -21011.411} C_VEL
LIN {X 0,Y 213.703,Z 287.405,A -85,B 0,C 180,E1 -21012.615,E2 -21012.615} C_VEL
LIN {X 0,Y 213.027,Z 286.115,A -85,B 0,C 180,E1 -21013.004,E2 -21013.004} C_VEL
LIN {X 0,Y 210.695,Z 282.747,A -85,B 0,C 180,E1 -21014.284,E2 -21014.284} C_VEL
LIN {X 0,Y 209.762,Z 280.047,A -85,B 0,C 180,E1 -21015,E2 -21015} C_VEL
LIN {X 0,Y 209.428,Z 278.076,A -85,B 0,C 180,E1 -21017.84,E2 -21017.84} C_VEL
LIN {X 0,Y 209.171,Z 276.298,A -85,B 0,C 180,E1 -21020.602,E2 -21020.602} C_VEL
LIN {X 0,Y 208.733,Z 273.791,A -85,B 0,C 180,E1 -21025.08,E2 -21025.08} C_VEL
LIN {X 0,Y 208.372,Z 271.688,A -85,B 0,C 180,E1 -21029.604,E2 -21029.604} C_VEL
LIN {X 0,Y 208.118,Z 270.087,A -85,B 0,C 180,E1 -21033.957,E2 -21033.957} C_VEL
LIN {X 0,Y 207.949,Z 268.937,A -85,B 0,C 180,E1 -21038.172,E2 -21038.172} C_VEL
LIN {X 0,Y 207.884,Z 268.177,A -85,B 0,C 180,E1 -21042.283,E2 -21042.283} C_VEL
LIN {X 0,Y 207.858,Z 267.764,A -85,B 0,C 180,E1 -21046.306,E2 -21046.306} C_VEL
LIN {X 0,Y 208.047,Z 267.63,A -85,B 0,C 180,E1 -21050.273,E2 -21050.273} C_VEL
LIN {X 0,Y 208.054,Z 267.847,A -85,B 0,C 180,E1 -21054.181,E2 -21054.181} C_VEL
LIN {X 0,Y 208.562,Z 268.582,A -85,B 0,C 180,E1 -21059.997,E2 -21059.997} C_VEL
LIN {X 0,Y 208.496,Z 269.066,A -85,B 0,C 180,E1 -21061.747,E2 -21061.747} C_VEL
LIN {X 0,Y 209.511,Z 271.7,A -85,B 0,C 180,E1 -21062.521,E2 -21062.521} C_VEL
LIN {X 0,Y 211.944,Z 274.534,A -85,B 0,C 180,E1 -21063.918,E2 -21063.918} C_VEL
LIN {X 0,Y 213.867,Z 277.921,A -85,B 0,C 180,E1 -21065.123,E2 -21065.123} C_VEL
LIN {X 0,Y 214.85,Z 278.932,A -85,B 0,C 180,E1 -21065.628,E2 -21065.628} C_VEL
LIN {X 0,Y 219.078,Z 287.047,A -85,B 0,C 180,E1 -21068.297,E2 -21068.297} C_VEL
LIN {X 0,Y 222.12,Z 294.503,A -85,B 0,C 180,E1 -21070.47,E2 -21070.47} C_VEL
LIN {X 0,Y 224.552,Z 302.58,A -85,B 0,C 180,E1 -21072.652,E2 -21072.652} C_VEL
LIN {X 0,Y 226.187,Z 311.15,A -85,B 0,C 180,E1 -21074.896,E2 -21074.896} C_VEL
LIN {X 0,Y 226.792,Z 317.975,A -85,B 0,C 180,E1 -21076.654,E2 -21076.654} C_VEL
LIN {X 0,Y 226.764,Z 319.791,A -85,B 0,C 180,E1 -21077.12,E2 -21077.12} C_VEL
LIN {X 0,Y 223.328,Z 329.855,A -85,B 0,C 180,E1 -21079.255,E2 -21079.255} C_VEL
LIN {X 0,Y 219.811,Z 338.717,A -85,B 0,C 180,E1 -21081.638,E2 -21081.638} C_VEL
LIN {X 0,Y 216.231,Z 347.013,A -85,B 0,C 180,E1 -21084.489,E2 -21084.489} C_VEL
LIN {X 0,Y 213.096,Z 353.721,A -85,B 0,C 180,E1 -21087.494,E2 -21087.494} C_VEL
LIN {X 0,Y 210.966,Z 358.033,A -85,B 0,C 180,E1 -21089.989,E2 -21089.989} C_VEL
LIN {X 0,Y 208.948,Z 361.752,A -85,B 0,C 180,E1 -21092.769,E2 -21092.769} C_VEL
LIN {X 0,Y 207.382,Z 364.479,A -85,B 0,C 180,E1 -21095.579,E2 -21095.579} C_VEL
LIN {X 0,Y 206.172,Z 366.301,A -85,B 0,C 180,E1 -21098.372,E2 -21098.372} C_VEL
LIN {X 0,Y 205.302,Z 367.288,A -85,B 0,C 180,E1 -21101.141,E2 -21101.141} C_VEL
LIN {X 0,Y 204.735,Z 367.501,A -85,B 0,C 180,E1 -21103.875,E2 -21103.875} C_VEL
LIN {X 0,Y 204.515,Z 366.921,A -85,B 0,C 180,E1 -21106.586,E2 -21106.586} C_VEL
LIN {X 0,Y 204.514,Z 365.626,A -85,B 0,C 180,E1 -21109.239,E2 -21109.239} C_VEL
LIN {X 0,Y 204.857,Z 363.412,A -85,B 0,C 180,E1 -21112.091,E2 -21112.091} C_VEL
LIN {X 0,Y 205.545,Z 360.02,A -85,B 0,C 180,E1 -21115.139,E2 -21115.139} C_VEL
LIN {X 0,Y 206.518,Z 355.275,A -85,B 0,C 180,E1 -21118.288,E2 -21118.288} C_VEL
LIN {X 0,Y 207.91,Z 348.965,A -85,B 0,C 180,E1 -21121.499,E2 -21121.499} C_VEL
LIN {X 0,Y 209.492,Z 342.37,A -85,B 0,C 180,E1 -21124.145,E2 -21124.145} C_VEL
LIN {X 0,Y 211.364,Z 333.967,A -85,B 0,C 180,E1 -21126.855,E2 -21126.855} C_VEL
LIN {X 0,Y 213.502,Z 324.594,A -85,B 0,C 180,E1 -21129.277,E2 -21129.277} C_VEL
LIN {X 0,Y 215.692,Z 313.989,A -85,B 0,C 180,E1 -21131.478,E2 -21131.478} C_VEL
LIN {X 0,Y 216.987,Z 306.19,A -85,B 0,C 180,E1 -21132.811,E2 -21132.811} C_VEL
LIN {X 0,Y 215.033,Z 294.581,A -85,B 0,C 180,E1 -21134.844,E2 -21134.844} C_VEL
LIN {X 0,Y 212.345,Z 282.831,A -85,B 0,C 180,E1 -21136.605,E2 -21136.605} C_VEL
LIN {X 0,Y 208.537,Z 269.817,A -85,B 0,C 180,E1 -21138.273,E2 -21138.273} C_VEL
LIN {X 0,Y 206.345,Z 262.799,A -85,B 0,C 180,E1 -21139.069,E2 -21139.069} C_VEL
LIN {X 0,Y 206.892,Z 262.715,A -85,B 0,C 180,E1 -21142.192,E2 -21142.192} C_VEL
LIN {X 0,Y 207.367,Z 262.657,A -85,B 0,C 180,E1 -21148.059,E2 -21148.059} C_VEL
LIN {X 0,Y 207.505,Z 262.639,A -85,B 0,C 180,E1 -21150.001,E2 -21150.001} C_VEL
LIN {X 0,Y 207.074,Z 262.69,A -85,B 0,C 180,E1 -21153.893,E2 -21153.893} C_VEL
LIN {X 0,Y 207.155,Z 262.68,A -85,B 0,C 180,E1 -21157.8,E2 -21157.8} C_VEL
LIN {X 0,Y 206.969,Z 262.699,A -85,B 0,C 180,E1 -21161.757,E2 -21161.757} C_VEL
LIN {X 0,Y 206.865,Z 262.719,A -85,B 0,C 180,E1 -21165.772,E2 -21165.772} C_VEL
LIN {X 0,Y 206.812,Z 262.723,A -85,B 0,C 180,E1 -21169.867,E2 -21169.867} C_VEL
LIN {X 0,Y 206.762,Z 262.731,A -85,B 0,C 180,E1 -21174.073,E2 -21174.073} C_VEL
LIN {X 0,Y 206.734,Z 262.73,A -85,B 0,C 180,E1 -21178.421,E2 -21178.421} C_VEL
LIN {X 0,Y 206.7,Z 262.738,A -85,B 0,C 180,E1 -21182.959,E2 -21182.959} C_VEL
LIN {X 0,Y 206.717,Z 262.728,A -85,B 0,C 180,E1 -21187.733,E2 -21187.733} C_VEL
LIN {X 0,Y 206.742,Z 262.731,A -85,B 0,C 180,E1 -21191.6,E2 -21191.6} C_VEL
LIN {X 0,Y 206.739,Z 262.725,A -85,B 0,C 180,E1 -21195.553,E2 -21195.553} C_VEL
LIN {X 0,Y 206.738,Z 262.726,A -85,B 0,C 180,E1 -21199.772,E2 -21199.772} C_VEL
LIN {X 0,Y 206.727,Z 262.733,A -85,B 0,C 180,E1 -21204.699,E2 -21204.699} C_VEL
LIN {X 0,Y 206.72,Z 262.721,A -85,B 0,C 180,E1 -21209.343,E2 -21209.343} C_VEL
LIN {X 0,Y 206.73,Z 262.73,A -85,B 0,C 180,E1 -21213.776,E2 -21213.776} C_VEL
LIN {X 0,Y 206.757,Z 262.73,A -85,B 0,C 180,E1 -21218.047,E2 -21218.047} C_VEL
LIN {X 0,Y 206.873,Z 262.702,A -85,B 0,C 180,E1 -21222.2,E2 -21222.2} C_VEL
LIN {X 0,Y 206.896,Z 262.711,A -85,B 0,C 180,E1 -21226.248,E2 -21226.248} C_VEL
LIN {X 0,Y 207.101,Z 262.687,A -85,B 0,C 180,E1 -21230.234,E2 -21230.234} C_VEL
LIN {X 0,Y 207.06,Z 262.681,A -85,B 0,C 180,E1 -21234.159,E2 -21234.159} C_VEL
LIN {X 0,Y 207.384,Z 262.649,A -85,B 0,C 180,E1 -21238.061,E2 -21238.061} C_VEL
LIN {X 0,Y 207.518,Z 262.636,A -85,B 0,C 180,E1 -21240.003,E2 -21240.003} C_VEL
LIN {X 0,Y 207.383,Z 262.653,A -85,B 0,C 180,E1 -21241.945,E2 -21241.945} C_VEL
LIN {X 0,Y 207.136,Z 262.675,A -85,B 0,C 180,E1 -21247.803,E2 -21247.803} C_VEL
LIN {X 0,Y 206.929,Z 262.71,A -85,B 0,C 180,E1 -21251.761,E2 -21251.761} C_VEL
LIN {X 0,Y 206.873,Z 262.709,A -85,B 0,C 180,E1 -21255.773,E2 -21255.773} C_VEL
LIN {X 0,Y 206.791,Z 262.726,A -85,B 0,C 180,E1 -21259.871,E2 -21259.871} C_VEL
LIN {X 0,Y 206.771,Z 262.728,A -85,B 0,C 180,E1 -21264.074,E2 -21264.074} C_VEL
LIN {X 0,Y 206.745,Z 262.731,A -85,B 0,C 180,E1 -21268.422,E2 -21268.422} C_VEL
LIN {X 0,Y 206.719,Z 262.736,A -85,B 0,C 180,E1 -21272.957,E2 -21272.957} C_VEL
LIN {X 0,Y 206.8,Z 262.902,A -85,B 0,C 180,E1 -21274.405,E2 -21274.405} C_VEL
LIN {X 0,Y 207.403,Z 266.55,A -85,B 0,C 180,E1 -21278.795,E2 -21278.795} C_VEL
LIN {X 0,Y 208.21,Z 270.934,A -85,B 0,C 180,E1 -21283.699,E2 -21283.699} C_VEL
LIN {X 0,Y 208.966,Z 274.721,A -85,B 0,C 180,E1 -21287.727,E2 -21287.727} C_VEL
LIN {X 0,Y 209.508,Z 278.69,A -85,B 0,C 180,E1 -21291.709,E2 -21291.709} C_VEL
LIN {X 0,Y 209.215,Z 280.84,A -85,B 0,C 180,E1 -21293.732,E2 -21293.732} C_VEL
LIN {X 0,Y 208.104,Z 285.186,A -85,B 0,C 180,E1 -21297.696,E2 -21297.696} C_VEL
LIN {X 0,Y 210.568,Z 299.183,A -85,B 0,C 180,E1 -21298.977,E2 -21298.977} C_VEL
LIN {X 0,Y 212.164,Z 311.41,A -85,B 0,C 180,E1 -21300.408,E2 -21300.408} C_VEL
LIN {X 0,Y 213.324,Z 324.356,A -85,B 0,C 180,E1 -21302.271,E2 -21302.271} C_VEL
LIN {X 0,Y 213.77,Z 335.569,A -85,B 0,C 180,E1 -21304.221,E2 -21304.221} C_VEL
LIN {X 0,Y 213.798,Z 343.034,A -85,B 0,C 180,E1 -21305.737,E2 -21305.737} C_VEL
LIN {X 0,Y 211.56,Z 353.252,A -85,B 0,C 180,E1 -21308.054,E2 -21308.054} C_VEL
LIN {X 0,Y 210.992,Z 355.788,A -85,B 0,C 180,E1 -21308.726,E2 -21308.726} C_VEL
LIN {X 0,Y 209.444,Z 359.808,A -85,B 0,C 180,E1 -21309.829,E2 -21309.829} C_VEL
LIN {X 0,Y 205.173,Z 365.795,A -85,B 0,C 180,E1 -21311.673,E2 -21311.673} C_VEL
LIN {X 0,Y 200.995,Z 371.161,A -85,B 0,C 180,E1 -21313.724,E2 -21313.724} C_VEL
LIN {X 0,Y 199.628,Z 374.21,A -85,B 0,C 180,E1 -21315.126,E2 -21315.126} C_VEL
LIN {X 0,Y 198.363,Z 380.706,A -85,B 0,C 180,E1 -21318.762,E2 -21318.762} C_VEL
LIN {X 0,Y 197.781,Z 384.819,A -85,B 0,C 180,E1 -21321.827,E2 -21321.827} C_VEL
LIN {X 0,Y 197.64,Z 387.676,A -85,B 0,C 180,E1 -21324.693,E2 -21324.693} C_VEL
LIN {X 0,Y 197.637,Z 389.868,A -85,B 0,C 180,E1 -21327.961,E2 -21327.961} C_VEL
LIN {X 0,Y 197.674,Z 390.695,A -85,B 0,C 180,E1 -21329.999,E2 -21329.999} C_VEL
LIN {X 0,Y 197.611,Z 391.083,A -85,B 0,C 180,E1 -21332.037,E2 -21332.037} C_VEL
LIN {X 0,Y 197.509,Z 390.621,A -85,B 0,C 180,E1 -21336.127,E2 -21336.127} C_VEL
LIN {X 0,Y 198.035,Z 388.629,A -85,B 0,C 180,E1 -21340.22,E2 -21340.22} C_VEL
LIN {X 0,Y 199.354,Z 384.976,A -85,B 0,C 180,E1 -21344.286,E2 -21344.286} C_VEL
LIN {X 0,Y 201.145,Z 381.144,A -85,B 0,C 180,E1 -21347.276,E2 -21347.276} C_VEL
LIN {X 0,Y 203.361,Z 376.264,A -85,B 0,C 180,E1 -21350.217,E2 -21350.217} C_VEL
LIN {X 0,Y 206.154,Z 370.122,A -85,B 0,C 180,E1 -21353.12,E2 -21353.12} C_VEL
LIN {X 0,Y 209.333,Z 362.772,A -85,B 0,C 180,E1 -21355.876,E2 -21355.876} C_VEL
LIN {X 0,Y 213.245,Z 353.647,A -85,B 0,C 180,E1 -21358.546,E2 -21358.546} C_VEL
LIN {X 0,Y 215.473,Z 344.594,A -85,B 0,C 180,E1 -21360.91,E2 -21360.91} C_VEL
LIN {X 0,Y 216.724,Z 335.105,A -85,B 0,C 180,E1 -21363.167,E2 -21363.167} C_VEL
LIN {X 0,Y 216.901,Z 323.888,A -85,B 0,C 180,E1 -21365.677,E2 -21365.677} C_VEL
LIN {X 0,Y 216.068,Z 313.697,A -85,B 0,C 180,E1 -21367.926,E2 -21367.926} C_VEL
LIN {X 0,Y 214.255,Z 303.979,A -85,B 0,C 180,E1 -21370.139,E2 -21370.139} C_VEL
LIN {X 0,Y 212.191,Z 297.718,A -85,B 0,C 180,E1 -21371.816,E2 -21371.816} C_VEL
LIN {X 0,Y 209.694,Z 292.179,A -85,B 0,C 180,E1 -21373.531,E2 -21373.531} C_VEL
LIN {X 0,Y 207.162,Z 287.987,A -85,B 0,C 180,E1 -21375.166,E2 -21375.166} C_VEL
LIN {X 0,Y 206.282,Z 285.759,A -85,B 0,C 180,E1 -21375.839,E2 -21375.839} C_VEL
LIN {X 0,Y 203.781,Z 282.661,A -85,B 0,C 180,E1 -21377.409,E2 -21377.409} C_VEL
LIN {X 0,Y 202.367,Z 279.024,A -85,B 0,C 180,E1 -21378.708,E2 -21378.708} C_VEL
LIN {X 0,Y 202.02,Z 276.434,A -85,B 0,C 180,E1 -21383.141,E2 -21383.141} C_VEL
LIN {X 0,Y 201.545,Z 273.872,A -85,B 0,C 180,E1 -21388.459,E2 -21388.459} C_VEL
LIN {X 0,Y 201.281,Z 272.15,A -85,B 0,C 180,E1 -21393.002,E2 -21393.002} C_VEL
LIN {X 0,Y 201.097,Z 270.892,A -85,B 0,C 180,E1 -21397.388,E2 -21397.388} C_VEL
LIN {X 0,Y 201.011,Z 270.027,A -85,B 0,C 180,E1 -21401.656,E2 -21401.656} C_VEL
LIN {X 0,Y 200.95,Z 269.546,A -85,B 0,C 180,E1 -21405.826,E2 -21405.826} C_VEL
LIN {X 0,Y 201.134,Z 269.352,A -85,B 0,C 180,E1 -21409.935,E2 -21409.935} C_VEL
LIN {X 0,Y 201.175,Z 269.512,A -85,B 0,C 180,E1 -21413.981,E2 -21413.981} C_VEL
LIN {X 0,Y 201.488,Z 270.064,A -85,B 0,C 180,E1 -21418.185,E2 -21418.185} C_VEL
LIN {X 0,Y 202.552,Z 272.403,A -85,B 0,C 180,E1 -21419.127,E2 -21419.127} C_VEL
LIN {X 0,Y 205.503,Z 275.634,A -85,B 0,C 180,E1 -21421.148,E2 -21421.148} C_VEL
LIN {X 0,Y 207.176,Z 278.802,A -85,B 0,C 180,E1 -21422.427,E2 -21422.427} C_VEL
LIN {X 0,Y 208.871,Z 281.257,A -85,B 0,C 180,E1 -21423.567,E2 -21423.567} C_VEL
LIN {X 0,Y 210.965,Z 284.463,A -85,B 0,C 180,E1 -21424.954,E2 -21424.954} C_VEL
LIN {X 0,Y 214.497,Z 291.637,A -85,B 0,C 180,E1 -21427.528,E2 -21427.528} C_VEL
LIN {X 0,Y 217.171,Z 298.774,A -85,B 0,C 180,E1 -21429.758,E2 -21429.758} C_VEL
LIN {X 0,Y 219.55,Z 308.16,A -85,B 0,C 180,E1 -21432.475,E2 -21432.475} C_VEL
LIN {X 0,Y 220.625,Z 316.354,A -85,B 0,C 180,E1 -21434.761,E2 -21434.761} C_VEL
LIN {X 0,Y 220.777,Z 321.666,A -85,B 0,C 180,E1 -21436.233,E2 -21436.233} C_VEL
LIN {X 0,Y 217.218,Z 331.342,A -85,B 0,C 180,E1 -21438.385,E2 -21438.385} C_VEL
LIN {X 0,Y 213.729,Z 339.663,A -85,B 0,C 180,E1 -21440.712,E2 -21440.712} C_VEL
LIN {X 0,Y 209.887,Z 347.995,A -85,B 0,C 180,E1 -21443.688,E2 -21443.688} C_VEL
LIN {X 0,Y 206.533,Z 354.593,A -85,B 0,C 180,E1 -21446.802,E2 -21446.802} C_VEL
LIN {X 0,Y 203.532,Z 360.149,A -85,B 0,C 180,E1 -21450.319,E2 -21450.319} C_VEL
LIN {X 0,Y 201.543,Z 363.443,A -85,B 0,C 180,E1 -21453.188,E2 -21453.188} C_VEL
LIN {X 0,Y 199.721,Z 366.215,A -85,B 0,C 180,E1 -21456.737,E2 -21456.737} C_VEL
LIN {X 0,Y 198.679,Z 367.452,A -85,B 0,C 180,E1 -21459.543,E2 -21459.543} C_VEL
LIN {X 0,Y 197.898,Z 367.948,A -85,B 0,C 180,E1 -21462.43,E2 -21462.43} C_VEL
LIN {X 0,Y 197.472,Z 367.645,A -85,B 0,C 180,E1 -21465.375,E2 -21465.375} C_VEL
LIN {X 0,Y 197.382,Z 366.477,A -85,B 0,C 180,E1 -21468.388,E2 -21468.388} C_VEL
LIN {X 0,Y 197.654,Z 364.357,A -85,B 0,C 180,E1 -21471.461,E2 -21471.461} C_VEL
LIN {X 0,Y 198.324,Z 361.188,A -85,B 0,C 180,E1 -21474.585,E2 -21474.585} C_VEL
LIN {X 0,Y 199.303,Z 356.315,A -85,B 0,C 180,E1 -21478.067,E2 -21478.067} C_VEL
LIN {X 0,Y 200.823,Z 349.696,A -85,B 0,C 180,E1 -21481.615,E2 -21481.615} C_VEL
LIN {X 0,Y 202.513,Z 342.914,A -85,B 0,C 180,E1 -21484.453,E2 -21484.453} C_VEL
LIN {X 0,Y 204.436,Z 334.564,A -85,B 0,C 180,E1 -21487.25,E2 -21487.25} C_VEL
LIN {X 0,Y 206.759,Z 324.734,A -85,B 0,C 180,E1 -21489.871,E2 -21489.871} C_VEL
LIN {X 0,Y 208.82,Z 315.063,A -85,B 0,C 180,E1 -21491.947,E2 -21491.947} C_VEL
LIN {X 0,Y 210.211,Z 307.777,A -85,B 0,C 180,E1 -21493.241,E2 -21493.241} C_VEL
LIN {X 0,Y 208.522,Z 297.042,A -85,B 0,C 180,E1 -21495.219,E2 -21495.219} C_VEL
LIN {X 0,Y 206.194,Z 286.288,A -85,B 0,C 180,E1 -21496.951,E2 -21496.951} C_VEL
LIN {X 0,Y 202.674,Z 273.565,A -85,B 0,C 180,E1 -21498.725,E2 -21498.725} C_VEL
LIN {X 0,Y 199.464,Z 263.652,A -85,B 0,C 180,E1 -21499.921,E2 -21499.921} C_VEL
LIN {X 0,Y 199.807,Z 263.598,A -85,B 0,C 180,E1 -21501.913,E2 -21501.913} C_VEL
LIN {X 0,Y 200.305,Z 263.537,A -85,B 0,C 180,E1 -21507.99,E2 -21507.99} C_VEL
LIN {X 0,Y 200.469,Z 263.515,A -85,B 0,C 180,E1 -21510.001,E2 -21510.001} C_VEL
LIN {X 0,Y 200.02,Z 263.569,A -85,B 0,C 180,E1 -21514.031,E2 -21514.031} C_VEL
LIN {X 0,Y 200.099,Z 263.559,A -85,B 0,C 180,E1 -21518.077,E2 -21518.077} C_VEL
LIN {X 0,Y 199.902,Z 263.579,A -85,B 0,C 180,E1 -21522.179,E2 -21522.179} C_VEL
LIN {X 0,Y 199.803,Z 263.599,A -85,B 0,C 180,E1 -21526.345,E2 -21526.345} C_VEL
LIN {X 0,Y 199.741,Z 263.605,A -85,B 0,C 180,E1 -21530.602,E2 -21530.602} C_VEL
LIN {X 0,Y 199.668,Z 263.613,A -85,B 0,C 180,E1 -21534.986,E2 -21534.986} C_VEL
LIN {X 0,Y 199.665,Z 263.614,A -85,B 0,C 180,E1 -21539.525,E2 -21539.525} C_VEL
LIN {X 0,Y 199.655,Z 263.617,A -85,B 0,C 180,E1 -21542.355,E2 -21542.355} C_VEL
LIN {X 0,Y 199.645,Z 263.607,A -85,B 0,C 180,E1 -21546.76,E2 -21546.76} C_VEL
LIN {X 0,Y 199.694,Z 263.608,A -85,B 0,C 180,E1 -21549.309,E2 -21549.309} C_VEL
LIN {X 0,Y 199.693,Z 263.611,A -85,B 0,C 180,E1 -21552.353,E2 -21552.353} C_VEL
LIN {X 0,Y 199.687,Z 263.604,A -85,B 0,C 180,E1 -21555.265,E2 -21555.265} C_VEL
LIN {X 0,Y 199.687,Z 263.597,A -85,B 0,C 180,E1 -21558.038,E2 -21558.038} C_VEL
LIN {X 0,Y 199.697,Z 263.608,A -85,B 0,C 180,E1 -21560.739,E2 -21560.739} C_VEL
LIN {X 0,Y 199.631,Z 263.616,A -85,B 0,C 180,E1 -21565.722,E2 -21565.722} C_VEL
LIN {X 0,Y 199.7,Z 263.6,A -85,B 0,C 180,E1 -21568.141,E2 -21568.141} C_VEL
LIN {X 0,Y 199.685,Z 263.607,A -85,B 0,C 180,E1 -21572.776,E2 -21572.776} C_VEL
LIN {X 0,Y 199.737,Z 263.603,A -85,B 0,C 180,E1 -21577.233,E2 -21577.233} C_VEL
LIN {X 0,Y 199.796,Z 263.585,A -85,B 0,C 180,E1 -21581.761,E2 -21581.761} C_VEL
LIN {X 0,Y 199.837,Z 263.586,A -85,B 0,C 180,E1 -21585.752,E2 -21585.752} C_VEL
LIN {X 0,Y 200.024,Z 263.57,A -85,B 0,C 180,E1 -21589.885,E2 -21589.885} C_VEL
LIN {X 0,Y 200.022,Z 263.559,A -85,B 0,C 180,E1 -21593.953,E2 -21593.953} C_VEL
LIN {X 0,Y 200.324,Z 263.527,A -85,B 0,C 180,E1 -21597.993,E2 -21597.993} C_VEL
LIN {X 0,Y 200.483,Z 263.512,A -85,B 0,C 180,E1 -21600.003,E2 -21600.003} C_VEL
LIN {X 0,Y 200.024,Z 263.565,A -85,B 0,C 180,E1 -21604.033,E2 -21604.033} C_VEL
LIN {X 0,Y 200.084,Z 263.556,A -85,B 0,C 180,E1 -21608.08,E2 -21608.08} C_VEL
LIN {X 0,Y 199.879,Z 263.586,A -85,B 0,C 180,E1 -21612.182,E2 -21612.182} C_VEL
LIN {X 0,Y 199.811,Z 263.587,A -85,B 0,C 180,E1 -21616.346,E2 -21616.346} C_VEL
LIN {X 0,Y 199.708,Z 263.607,A -85,B 0,C 180,E1 -21620.608,E2 -21620.608} C_VEL
LIN {X 0,Y 199.681,Z 263.612,A -85,B 0,C 180,E1 -21624.987,E2 -21624.987} C_VEL
LIN {X 0,Y 199.673,Z 263.614,A -85,B 0,C 180,E1 -21629.526,E2 -21629.526} C_VEL
LIN {X 0,Y 199.717,Z 263.671,A -85,B 0,C 180,E1 -21633.738,E2 -21633.738} C_VEL
LIN {X 0,Y 200.272,Z 266.972,A -85,B 0,C 180,E1 -21637.891,E2 -21637.891} C_VEL
LIN {X 0,Y 201.031,Z 271.127,A -85,B 0,C 180,E1 -21642.763,E2 -21642.763} C_VEL
LIN {X 0,Y 201.785,Z 274.968,A -85,B 0,C 180,E1 -21647.009,E2 -21647.009} C_VEL
LIN {X 0,Y 202.285,Z 277.652,A -85,B 0,C 180,E1 -21649.853,E2 -21649.853} C_VEL
LIN {X 0,Y 202.439,Z 279.086,A -85,B 0,C 180,E1 -21651.324,E2 -21651.324} C_VEL
LIN {X 0,Y 202.109,Z 281.592,A -85,B 0,C 180,E1 -21653.76,E2 -21653.76} C_VEL
LIN {X 0,Y 201.244,Z 284.785,A -85,B 0,C 180,E1 -21656.788,E2 -21656.788} C_VEL
LIN {X 0,Y 203.707,Z 298.676,A -85,B 0,C 180,E1 -21658.14,E2 -21658.14} C_VEL
LIN {X 0,Y 205.343,Z 311.686,A -85,B 0,C 180,E1 -21659.727,E2 -21659.727} C_VEL
LIN {X 0,Y 206.414,Z 323.775,A -85,B 0,C 180,E1 -21661.531,E2 -21661.531} C_VEL
LIN {X 0,Y 206.842,Z 334.246,A -85,B 0,C 180,E1 -21663.391,E2 -21663.391} C_VEL
LIN {X 0,Y 206.797,Z 343.799,A -85,B 0,C 180,E1 -21665.397,E2 -21665.397} C_VEL
LIN {X 0,Y 204.516,Z 353.745,A -85,B 0,C 180,E1 -21667.789,E2 -21667.789} C_VEL
LIN {X 0,Y 202.57,Z 361.925,A -85,B 0,C 180,E1 -21670.228,E2 -21670.228} C_VEL
LIN {X 0,Y 200.646,Z 369.953,A -85,B 0,C 180,E1 -21673.203,E2 -21673.203} C_VEL
LIN {X 0,Y 199.628,Z 374.21,A -85,B 0,C 180,E1 -21675.126,E2 -21675.126} C_VEL
LIN {X 0,Y 198.359,Z 377.041,A -85,B 0,C 180,E1 -21676.58,E2 -21676.58} C_VEL
LIN {X 0,Y 194.709,Z 380.978,A -85,B 0,C 180,E1 -21679.018,E2 -21679.018} C_VEL
LIN {X 0,Y 191.883,Z 383.598,A -85,B 0,C 180,E1 -21681.087,E2 -21681.087} C_VEL
LIN {X 0,Y 190.696,Z 385.385,A -85,B 0,C 180,E1 -21682.745,E2 -21682.745} C_VEL
LIN {X 0,Y 190.598,Z 385.937,A -85,B 0,C 180,E1 -21683.313,E2 -21683.313} C_VEL
LIN {X 0,Y 190.541,Z 388,A -85,B 0,C 180,E1 -21685.768,E2 -21685.768} C_VEL
LIN {X 0,Y 190.574,Z 389.285,A -85,B 0,C 180,E1 -21687.885,E2 -21687.885} C_VEL
LIN {X 0,Y 190.609,Z 390.154,A -85,B 0,C 180,E1 -21689.999,E2 -21689.999} C_VEL
LIN {X 0,Y 190.519,Z 390.61,A -85,B 0,C 180,E1 -21692.113,E2 -21692.113} C_VEL
LIN {X 0,Y 190.437,Z 390.554,A -85,B 0,C 180,E1 -21694.816,E2 -21694.816} C_VEL
LIN {X 0,Y 190.623,Z 389.487,A -85,B 0,C 180,E1 -21698.479,E2 -21698.479} C_VEL
LIN {X 0,Y 191.636,Z 386.822,A -85,B 0,C 180,E1 -21702.71,E2 -21702.71} C_VEL
LIN {X 0,Y 193.024,Z 383.741,A -85,B 0,C 180,E1 -21705.846,E2 -21705.846} C_VEL
LIN {X 0,Y 195.116,Z 379.672,A -85,B 0,C 180,E1 -21708.914,E2 -21708.914} C_VEL
LIN {X 0,Y 197.696,Z 374.532,A -85,B 0,C 180,E1 -21711.916,E2 -21711.916} C_VEL
LIN {X 0,Y 201.164,Z 366.982,A -85,B 0,C 180,E1 -21715.338,E2 -21715.338} C_VEL
LIN {X 0,Y 204.969,Z 358.962,A -85,B 0,C 180,E1 -21718.128,E2 -21718.128} C_VEL
LIN {X 0,Y 207.624,Z 352.651,A -85,B 0,C 180,E1 -21719.951,E2 -21719.951} C_VEL
LIN {X 0,Y 209.809,Z 343.566,A -85,B 0,C 180,E1 -21722.407,E2 -21722.407} C_VEL
LIN {X 0,Y 210.976,Z 333.721,A -85,B 0,C 180,E1 -21724.867,E2 -21724.867} C_VEL
LIN {X 0,Y 211.225,Z 324.774,A -85,B 0,C 180,E1 -21727.005,E2 -21727.005} C_VEL
LIN {X 0,Y 210.624,Z 315.863,A -85,B 0,C 180,E1 -21729.12,E2 -21729.12} C_VEL
LIN {X 0,Y 209.626,Z 308.776,A -85,B 0,C 180,E1 -21730.846,E2 -21730.846} C_VEL
LIN {X 0,Y 207.957,Z 302.831,A -85,B 0,C 180,E1 -21732.523,E2 -21732.523} C_VEL
LIN {X 0,Y 205.897,Z 297.799,A -85,B 0,C 180,E1 -21734.205,E2 -21734.205} C_VEL
LIN {X 0,Y 203.255,Z 292.565,A -85,B 0,C 180,E1 -21736.244,E2 -21736.244} C_VEL
LIN {X 0,Y 202.568,Z 291.256,A -85,B 0,C 180,E1 -21736.766,E2 -21736.766} C_VEL
LIN {X 0,Y 200.345,Z 287.644,A -85,B 0,C 180,E1 -21738.495,E2 -21738.495} C_VEL
LIN {X 0,Y 199.297,Z 285.052,A -85,B 0,C 180,E1 -21739.492,E2 -21739.492} C_VEL
LIN {X 0,Y 196.397,Z 281.405,A -85,B 0,C 180,E1 -21741.88,E2 -21741.88} C_VEL
LIN {X 0,Y 195.174,Z 278.254,A -85,B 0,C 180,E1 -21743.271,E2 -21743.271} C_VEL
LIN {X 0,Y 195.072,Z 277.87,A -85,B 0,C 180,E1 -21743.522,E2 -21743.522} C_VEL
LIN {X 0,Y 194.745,Z 276.076,A -85,B 0,C 180,E1 -21747.223,E2 -21747.223} C_VEL
LIN {X 0,Y 194.421,Z 274.238,A -85,B 0,C 180,E1 -21751.967,E2 -21751.967} C_VEL
LIN {X 0,Y 194.225,Z 272.876,A -85,B 0,C 180,E1 -21756.541,E2 -21756.541} C_VEL
LIN {X 0,Y 194.138,Z 271.907,A -85,B 0,C 180,E1 -21760.982,E2 -21760.982} C_VEL
LIN {X 0,Y 194.053,Z 271.366,A -85,B 0,C 180,E1 -21765.311,E2 -21765.311} C_VEL
LIN {X 0,Y 194.223,Z 271.109,A -85,B 0,C 180,E1 -21769.573,E2 -21769.573} C_VEL
LIN {X 0,Y 194.298,Z 271.313,A -85,B 0,C 180,E1 -21773.311,E2 -21773.311} C_VEL
LIN {X 0,Y 195.594,Z 273.989,A -85,B 0,C 180,E1 -21774.843,E2 -21774.843} C_VEL
LIN {X 0,Y 198.212,Z 276.202,A -85,B 0,C 180,E1 -21777.126,E2 -21777.126} C_VEL
LIN {X 0,Y 198.929,Z 276.912,A -85,B 0,C 180,E1 -21777.693,E2 -21777.693} C_VEL
LIN {X 0,Y 200.651,Z 279.738,A -85,B 0,C 180,E1 -21779.244,E2 -21779.244} C_VEL
LIN {X 0,Y 202.417,Z 282.087,A -85,B 0,C 180,E1 -21780.65,E2 -21780.65} C_VEL
LIN {X 0,Y 205.26,Z 286.947,A -85,B 0,C 180,E1 -21782.941,E2 -21782.941} C_VEL
LIN {X 0,Y 207.815,Z 291.763,A -85,B 0,C 180,E1 -21785.005,E2 -21785.005} C_VEL
LIN {X 0,Y 210.369,Z 297.522,A -85,B 0,C 180,E1 -21787.194,E2 -21787.194} C_VEL
LIN {X 0,Y 212.575,Z 304.507,A -85,B 0,C 180,E1 -21789.512,E2 -21789.512} C_VEL
LIN {X 0,Y 214.094,Z 311.989,A -85,B 0,C 180,E1 -21791.836,E2 -21791.836} C_VEL
LIN {X 0,Y 214.83,Z 319.919,A -85,B 0,C 180,E1 -21794.199,E2 -21794.199} C_VEL
LIN {X 0,Y 214.873,Z 323.168,A -85,B 0,C 180,E1 -21795.165,E2 -21795.165} C_VEL
LIN {X 0,Y 213.03,Z 328.424,A -85,B 0,C 180,E1 -21796.375,E2 -21796.375} C_VEL
LIN {X 0,Y 209.082,Z 337.567,A -85,B 0,C 180,E1 -21798.776,E2 -21798.776} C_VEL
LIN {X 0,Y 205.358,Z 345.513,A -85,B 0,C 180,E1 -21801.436,E2 -21801.436} C_VEL
LIN {X 0,Y 202.08,Z 351.821,A -85,B 0,C 180,E1 -21804.116,E2 -21804.116} C_VEL
LIN {X 0,Y 198.461,Z 358.214,A -85,B 0,C 180,E1 -21807.713,E2 -21807.713} C_VEL
LIN {X 0,Y 196.073,Z 362.097,A -85,B 0,C 180,E1 -21810.658,E2 -21810.658} C_VEL
LIN {X 0,Y 194.15,Z 364.987,A -85,B 0,C 180,E1 -21813.639,E2 -21813.639} C_VEL
LIN {X 0,Y 192.661,Z 366.969,A -85,B 0,C 180,E1 -21816.63,E2 -21816.63} C_VEL
LIN {X 0,Y 191.568,Z 368.105,A -85,B 0,C 180,E1 -21819.61,E2 -21819.61} C_VEL
LIN {X 0,Y 190.794,Z 368.413,A -85,B 0,C 180,E1 -21822.55,E2 -21822.55} C_VEL
LIN {X 0,Y 190.371,Z 367.972,A -85,B 0,C 180,E1 -21825.46,E2 -21825.46} C_VEL
LIN {X 0,Y 190.294,Z 366.821,A -85,B 0,C 180,E1 -21828.336,E2 -21828.336} C_VEL
LIN {X 0,Y 190.756,Z 363.719,A -85,B 0,C 180,E1 -21832.563,E2 -21832.563} C_VEL
LIN {X 0,Y 191.762,Z 359.02,A -85,B 0,C 180,E1 -21836.652,E2 -21836.652} C_VEL
LIN {X 0,Y 193.001,Z 353.548,A -85,B 0,C 180,E1 -21840.101,E2 -21840.101} C_VEL
LIN {X 0,Y 194.498,Z 347.422,A -85,B 0,C 180,E1 -21843.119,E2 -21843.119} C_VEL
LIN {X 0,Y 196.475,Z 339.375,A -85,B 0,C 180,E1 -21846.272,E2 -21846.272} C_VEL
LIN {X 0,Y 198.685,Z 330.448,A -85,B 0,C 180,E1 -21849.029,E2 -21849.029} C_VEL
LIN {X 0,Y 201.167,Z 319.706,A -85,B 0,C 180,E1 -21851.675,E2 -21851.675} C_VEL
LIN {X 0,Y 203.349,Z 309.298,A -85,B 0,C 180,E1 -21853.693,E2 -21853.693} C_VEL
LIN {X 0,Y 202.199,Z 300.557,A -85,B 0,C 180,E1 -21855.406,E2 -21855.406} C_VEL
LIN {X 0,Y 200.009,Z 289.744,A -85,B 0,C 180,E1 -21857.291,E2 -21857.291} C_VEL
LIN {X 0,Y 197.022,Z 278.297,A -85,B 0,C 180,E1 -21859.044,E2 -21859.044} C_VEL
LIN {X 0,Y 193.348,Z 266.984,A -85,B 0,C 180,E1 -21860.556,E2 -21860.556} C_VEL
LIN {X 0,Y 192.597,Z 264.495,A -85,B 0,C 180,E1 -21860.878,E2 -21860.878} C_VEL
LIN {X 0,Y 192.865,Z 264.464,A -85,B 0,C 180,E1 -21863.725,E2 -21863.725} C_VEL
LIN {X 0,Y 193.245,Z 264.417,A -85,B 0,C 180,E1 -21867.917,E2 -21867.917} C_VEL
LIN {X 0,Y 193.432,Z 264.392,A -85,B 0,C 180,E1 -21870.001,E2 -21870.001} C_VEL
LIN {X 0,Y 192.966,Z 264.448,A -85,B 0,C 180,E1 -21874.178,E2 -21874.178} C_VEL
LIN {X 0,Y 193.049,Z 264.437,A -85,B 0,C 180,E1 -21878.374,E2 -21878.374} C_VEL
LIN {X 0,Y 192.841,Z 264.46,A -85,B 0,C 180,E1 -21882.632,E2 -21882.632} C_VEL
LIN {X 0,Y 192.771,Z 264.47,A -85,B 0,C 180,E1 -21888.589,E2 -21888.589} C_VEL
LIN {X 0,Y 192.662,Z 264.489,A -85,B 0,C 180,E1 -21894.233,E2 -21894.233} C_VEL
LIN {X 0,Y 192.64,Z 264.488,A -85,B 0,C 180,E1 -21898.895,E2 -21898.895} C_VEL
LIN {X 0,Y 192.591,Z 264.494,A -85,B 0,C 180,E1 -21903.188,E2 -21903.188} C_VEL
LIN {X 0,Y 192.605,Z 264.487,A -85,B 0,C 180,E1 -21908.341,E2 -21908.341} C_VEL
LIN {X 0,Y 192.626,Z 264.488,A -85,B 0,C 180,E1 -21913.144,E2 -21913.144} C_VEL
LIN {X 0,Y 192.621,Z 264.476,A -85,B 0,C 180,E1 -21916.864,E2 -21916.864} C_VEL
LIN {X 0,Y 192.608,Z 264.49,A -85,B 0,C 180,E1 -21921.667,E2 -21921.667} C_VEL
LIN {X 0,Y 192.597,Z 264.488,A -85,B 0,C 180,E1 -21926.819,E2 -21926.819} C_VEL
LIN {X 0,Y 192.662,Z 264.475,A -85,B 0,C 180,E1 -21931.696,E2 -21931.696} C_VEL
LIN {X 0,Y 192.704,Z 264.481,A -85,B 0,C 180,E1 -21936.353,E2 -21936.353} C_VEL
LIN {X 0,Y 192.732,Z 264.467,A -85,B 0,C 180,E1 -21941.461,E2 -21941.461} C_VEL
LIN {X 0,Y 192.765,Z 264.465,A -85,B 0,C 180,E1 -21945.218,E2 -21945.218} C_VEL
LIN {X 0,Y 192.947,Z 264.451,A -85,B 0,C 180,E1 -21949.57,E2 -21949.57} C_VEL
LIN {X 0,Y 192.984,Z 264.436,A -85,B 0,C 180,E1 -21953.731,E2 -21953.731} C_VEL
LIN {X 0,Y 193.265,Z 264.405,A -85,B 0,C 180,E1 -21957.92,E2 -21957.92} C_VEL
LIN {X 0,Y 193.447,Z 264.389,A -85,B 0,C 180,E1 -21960.003,E2 -21960.003} C_VEL
LIN {X 0,Y 192.969,Z 264.443,A -85,B 0,C 180,E1 -21964.181,E2 -21964.181} C_VEL
LIN {X 0,Y 193.033,Z 264.434,A -85,B 0,C 180,E1 -21968.377,E2 -21968.377} C_VEL
LIN {X 0,Y 192.807,Z 264.467,A -85,B 0,C 180,E1 -21972.636,E2 -21972.636} C_VEL
LIN {X 0,Y 192.764,Z 264.465,A -85,B 0,C 180,E1 -21976.961,E2 -21976.961} C_VEL
LIN {X 0,Y 192.645,Z 264.489,A -85,B 0,C 180,E1 -21981.4,E2 -21981.4} C_VEL
LIN {X 0,Y 192.672,Z 264.484,A -85,B 0,C 180,E1 -21984.227,E2 -21984.227} C_VEL
LIN {X 0,Y 192.652,Z 264.488,A -85,B 0,C 180,E1 -21988.891,E2 -21988.891} C_VEL
LIN {X 0,Y 192.682,Z 264.507,A -85,B 0,C 180,E1 -21993.173,E2 -21993.173} C_VEL
LIN {X 0,Y 193.315,Z 268.373,A -85,B 0,C 180,E1 -21998.177,E2 -21998.177} C_VEL
LIN {X 0,Y 194.124,Z 272.894,A -85,B 0,C 180,E1 -22003.607,E2 -22003.607} C_VEL
LIN {X 0,Y 194.884,Z 276.589,A -85,B 0,C 180,E1 -22007.813,E2 -22007.813} C_VEL
LIN {X 0,Y 195.346,Z 279.525,A -85,B 0,C 180,E1 -22010.978,E2 -22010.978} C_VEL
LIN {X 0,Y 195.075,Z 282.074,A -85,B 0,C 180,E1 -22013.571,E2 -22013.571} C_VEL
LIN {X 0,Y 194.422,Z 284.596,A -85,B 0,C 180,E1 -22015.867,E2 -22015.867} C_VEL
LIN {X 0,Y 196.778,Z 297.836,A -85,B 0,C 180,E1 -22017.198,E2 -22017.198} C_VEL
LIN {X 0,Y 198.367,Z 310.114,A -85,B 0,C 180,E1 -22018.747,E2 -22018.747} C_VEL
LIN {X 0,Y 199.46,Z 322.53,A -85,B 0,C 180,E1 -22020.65,E2 -22020.65} C_VEL
LIN {X 0,Y 199.932,Z 334.261,A -85,B 0,C 180,E1 -22022.807,E2 -22022.807} C_VEL
LIN {X 0,Y 199.819,Z 344.371,A -85,B 0,C 180,E1 -22025.034,E2 -22025.034} C_VEL
LIN {X 0,Y 197.42,Z 354.242,A -85,B 0,C 180,E1 -22027.533,E2 -22027.533} C_VEL
LIN {X 0,Y 195.505,Z 362.183,A -85,B 0,C 180,E1 -22030.03,E2 -22030.03} C_VEL
LIN {X 0,Y 193.519,Z 370.076,A -85,B 0,C 180,E1 -22033.109,E2 -22033.109} C_VEL
LIN {X 0,Y 192.002,Z 376.366,A -85,B 0,C 180,E1 -22036.235,E2 -22036.235} C_VEL
LIN {X 0,Y 191.142,Z 381.374,A -85,B 0,C 180,E1 -22039.405,E2 -22039.405} C_VEL
LIN {X 0,Y 190.598,Z 385.937,A -85,B 0,C 180,E1 -22043.313,E2 -22043.313} C_VEL
LIN {X 0,Y 189.924,Z 387.439,A -85,B 0,C 180,E1 -22045.02,E2 -22045.02} C_VEL
LIN {X 0,Y 188.353,Z 388.561,A -85,B 0,C 180,E1 -22046.723,E2 -22046.723} C_VEL
LIN {X 0,Y 184.621,Z 389.838,A -85,B 0,C 180,E1 -22050.22,E2 -22050.22} C_VEL
LIN {X 0,Y 183.388,Z 390.132,A -85,B 0,C 180,E1 -22052.686,E2 -22052.686} C_VEL
LIN {X 0,Y 183.364,Z 389.881,A -85,B 0,C 180,E1 -22056.601,E2 -22056.601} C_VEL
LIN {X 0,Y 184.015,Z 388.085,A -85,B 0,C 180,E1 -22061.008,E2 -22061.008} C_VEL
LIN {X 0,Y 184.673,Z 386.618,A -85,B 0,C 180,E1 -22063.198,E2 -22063.198} C_VEL
LIN {X 0,Y 186.181,Z 383.624,A -85,B 0,C 180,E1 -22066.445,E2 -22066.445} C_VEL
LIN {X 0,Y 188.366,Z 379.664,A -85,B 0,C 180,E1 -22069.619,E2 -22069.619} C_VEL
LIN {X 0,Y 191.113,Z 374.671,A -85,B 0,C 180,E1 -22072.712,E2 -22072.712} C_VEL
LIN {X 0,Y 194.778,Z 367.366,A -85,B 0,C 180,E1 -22076.231,E2 -22076.231} C_VEL
LIN {X 0,Y 198.773,Z 359.509,A -85,B 0,C 180,E1 -22079.087,E2 -22079.087} C_VEL
LIN {X 0,Y 201.482,Z 353.371,A -85,B 0,C 180,E1 -22080.963,E2 -22080.963} C_VEL
LIN {X 0,Y 203.83,Z 344.596,A -85,B 0,C 180,E1 -22083.481,E2 -22083.481} C_VEL
LIN {X 0,Y 205.222,Z 335.144,A -85,B 0,C 180,E1 -22085.999,E2 -22085.999} C_VEL
LIN {X 0,Y 205.652,Z 325.531,A -85,B 0,C 180,E1 -22088.437,E2 -22088.437} C_VEL
LIN {X 0,Y 205.263,Z 317.161,A -85,B 0,C 180,E1 -22090.581,E2 -22090.581} C_VEL
LIN {X 0,Y 204.271,Z 310.335,A -85,B 0,C 180,E1 -22092.444,E2 -22092.444} C_VEL
LIN {X 0,Y 202.224,Z 304.183,A -85,B 0,C 180,E1 -22094.56,E2 -22094.56} C_VEL
LIN {X 0,Y 199.265,Z 297.233,A -85,B 0,C 180,E1 -22097.313,E2 -22097.313} C_VEL
LIN {X 0,Y 196.984,Z 293.138,A -85,B 0,C 180,E1 -22099.364,E2 -22099.364} C_VEL
LIN {X 0,Y 196.098,Z 290.933,A -85,B 0,C 180,E1 -22100.325,E2 -22100.325} C_VEL
LIN {X 0,Y 193.514,Z 287.03,A -85,B 0,C 180,E1 -22102.855,E2 -22102.855} C_VEL
LIN {X 0,Y 192.476,Z 284.198,A -85,B 0,C 180,E1 -22104.249,E2 -22104.249} C_VEL
LIN {X 0,Y 188.442,Z 278.696,A -85,B 0,C 180,E1 -22109.741,E2 -22109.741} C_VEL
LIN {X 0,Y 187.537,Z 275.934,A -85,B 0,C 180,E1 -22112.063,E2 -22112.063} C_VEL
LIN {X 0,Y 187.371,Z 274.869,A -85,B 0,C 180,E1 -22115.629,E2 -22115.629} C_VEL
LIN {X 0,Y 187.228,Z 273.805,A -85,B 0,C 180,E1 -22120.252,E2 -22120.252} C_VEL
LIN {X 0,Y 187.196,Z 273.279,A -85,B 0,C 180,E1 -22124.621,E2 -22124.621} C_VEL
LIN {X 0,Y 189.102,Z 276.087,A -85,B 0,C 180,E1 -22129,E2 -22129} C_VEL
LIN {X 0,Y 192.119,Z 278.123,A -85,B 0,C 180,E1 -22132.825,E2 -22132.825} C_VEL
LIN {X 0,Y 193.591,Z 280.964,A -85,B 0,C 180,E1 -22134.789,E2 -22134.789} C_VEL
LIN {X 0,Y 195.896,Z 282.867,A -85,B 0,C 180,E1 -22136.925,E2 -22136.925} C_VEL
LIN {X 0,Y 199.045,Z 287.908,A -85,B 0,C 180,E1 -22139.997,E2 -22139.997} C_VEL
LIN {X 0,Y 203.25,Z 296.007,A -85,B 0,C 180,E1 -22143.962,E2 -22143.962} C_VEL
LIN {X 0,Y 205.613,Z 301.894,A -85,B 0,C 180,E1 -22146.368,E2 -22146.368} C_VEL
LIN {X 0,Y 207.481,Z 308.813,A -85,B 0,C 180,E1 -22148.859,E2 -22148.859} C_VEL
LIN {X 0,Y 208.632,Z 315.783,A -85,B 0,C 180,E1 -22151.165,E2 -22151.165} C_VEL
LIN {X 0,Y 209.001,Z 323.384,A -85,B 0,C 180,E1 -22153.611,E2 -22153.611} C_VEL
LIN {X 0,Y 208.908,Z 325.734,A -85,B 0,C 180,E1 -22154.362,E2 -22154.362} C_VEL
LIN {X 0,Y 204.796,Z 335.349,A -85,B 0,C 180,E1 -22156.744,E2 -22156.744} C_VEL
LIN {X 0,Y 200.951,Z 343.212,A -85,B 0,C 180,E1 -22159.219,E2 -22159.219} C_VEL
LIN {X 0,Y 197.151,Z 350.272,A -85,B 0,C 180,E1 -22162.056,E2 -22162.056} C_VEL
LIN {X 0,Y 193.825,Z 355.955,A -85,B 0,C 180,E1 -22164.979,E2 -22164.979} C_VEL
LIN {X 0,Y 190.442,Z 361.344,A -85,B 0,C 180,E1 -22168.664,E2 -22168.664} C_VEL
LIN {X 0,Y 187.501,Z 365.441,A -85,B 0,C 180,E1 -22172.791,E2 -22172.791} C_VEL
LIN {X 0,Y 185.303,Z 368.012,A -85,B 0,C 180,E1 -22177.208,E2 -22177.208} C_VEL
LIN {X 0,Y 184.194,Z 368.798,A -85,B 0,C 180,E1 -22180.434,E2 -22180.434} C_VEL
LIN {X 0,Y 183.498,Z 368.737,A -85,B 0,C 180,E1 -22183.577,E2 -22183.577} C_VEL
LIN {X 0,Y 183.201,Z 367.849,A -85,B 0,C 180,E1 -22186.787,E2 -22186.787} C_VEL
LIN {X 0,Y 183.283,Z 366.06,A -85,B 0,C 180,E1 -22190.07,E2 -22190.07} C_VEL
LIN {X 0,Y 183.817,Z 363.281,A -85,B 0,C 180,E1 -22193.401,E2 -22193.401} C_VEL
LIN {X 0,Y 184.699,Z 359.311,A -85,B 0,C 180,E1 -22196.83,E2 -22196.83} C_VEL
LIN {X 0,Y 186.061,Z 353.491,A -85,B 0,C 180,E1 -22200.592,E2 -22200.592} C_VEL
LIN {X 0,Y 187.785,Z 346.828,A -85,B 0,C 180,E1 -22203.915,E2 -22203.915} C_VEL
LIN {X 0,Y 189.926,Z 338.332,A -85,B 0,C 180,E1 -22207.217,E2 -22207.217} C_VEL
LIN {X 0,Y 192.21,Z 329.474,A -85,B 0,C 180,E1 -22209.954,E2 -22209.954} C_VEL
LIN {X 0,Y 194.505,Z 319.704,A -85,B 0,C 180,E1 -22212.387,E2 -22212.387} C_VEL
LIN {X 0,Y 196.472,Z 310.831,A -85,B 0,C 180,E1 -22214.173,E2 -22214.173} C_VEL
LIN {X 0,Y 196.251,Z 307.041,A -85,B 0,C 180,E1 -22214.953,E2 -22214.953} C_VEL
LIN {X 0,Y 194.603,Z 296.871,A -85,B 0,C 180,E1 -22216.956,E2 -22216.956} C_VEL
LIN {X 0,Y 191.841,Z 284.958,A -85,B 0,C 180,E1 -22219.003,E2 -22219.003} C_VEL
LIN {X 0,Y 188.13,Z 272.366,A -85,B 0,C 180,E1 -22220.889,E2 -22220.889} C_VEL
LIN {X 0,Y 185.667,Z 265.36,A -85,B 0,C 180,E1 -22221.909,E2 -22221.909} C_VEL
LIN {X 0,Y 186.187,Z 265.296,A -85,B 0,C 180,E1 -22227.838,E2 -22227.838} C_VEL
LIN {X 0,Y 186.395,Z 265.269,A -85,B 0,C 180,E1 -22230.001,E2 -22230.001} C_VEL
LIN {X 0,Y 185.914,Z 265.326,A -85,B 0,C 180,E1 -22234.337,E2 -22234.337} C_VEL
LIN {X 0,Y 185.996,Z 265.317,A -85,B 0,C 180,E1 -22238.694,E2 -22238.694} C_VEL
LIN {X 0,Y 185.754,Z 265.346,A -85,B 0,C 180,E1 -22243.122,E2 -22243.122} C_VEL
LIN {X 0,Y 185.709,Z 265.351,A -85,B 0,C 180,E1 -22247.624,E2 -22247.624} C_VEL
LIN {X 0,Y 185.612,Z 265.368,A -85,B 0,C 180,E1 -22252.251,E2 -22252.251} C_VEL
LIN {X 0,Y 185.554,Z 265.366,A -85,B 0,C 180,E1 -22257.035,E2 -22257.035} C_VEL
LIN {X 0,Y 185.569,Z 265.37,A -85,B 0,C 180,E1 -22259.496,E2 -22259.496} C_VEL
LIN {X 0,Y 185.512,Z 265.371,A -85,B 0,C 180,E1 -22264.631,E2 -22264.631} C_VEL
LIN {X 0,Y 185.56,Z 265.363,A -85,B 0,C 180,E1 -22267.317,E2 -22267.317} C_VEL
LIN {X 0,Y 185.577,Z 265.37,A -85,B 0,C 180,E1 -22270.769,E2 -22270.769} C_VEL
LIN {X 0,Y 185.579,Z 265.359,A -85,B 0,C 180,E1 -22276.018,E2 -22276.018} C_VEL
LIN {X 0,Y 185.56,Z 265.363,A -85,B 0,C 180,E1 -22279.925,E2 -22279.925} C_VEL
LIN {X 0,Y 185.571,Z 265.37,A -85,B 0,C 180,E1 -22282.707,E2 -22282.707} C_VEL
LIN {X 0,Y 185.542,Z 265.363,A -85,B 0,C 180,E1 -22287.979,E2 -22287.979} C_VEL
LIN {X 0,Y 185.579,Z 265.354,A -85,B 0,C 180,E1 -22290.58,E2 -22290.58} C_VEL
LIN {X 0,Y 185.586,Z 265.365,A -85,B 0,C 180,E1 -22295.387,E2 -22295.387} C_VEL
LIN {X 0,Y 185.675,Z 265.345,A -85,B 0,C 180,E1 -22301.137,E2 -22301.137} C_VEL
LIN {X 0,Y 185.696,Z 265.345,A -85,B 0,C 180,E1 -22304.641,E2 -22304.641} C_VEL
LIN {X 0,Y 185.89,Z 265.329,A -85,B 0,C 180,E1 -22309.422,E2 -22309.422} C_VEL
LIN {X 0,Y 185.947,Z 265.314,A -85,B 0,C 180,E1 -22313.493,E2 -22313.493} C_VEL
LIN {X 0,Y 186.209,Z 265.283,A -85,B 0,C 180,E1 -22317.841,E2 -22317.841} C_VEL
LIN {X 0,Y 186.41,Z 265.265,A -85,B 0,C 180,E1 -22320.004,E2 -22320.004} C_VEL
LIN {X 0,Y 185.916,Z 265.321,A -85,B 0,C 180,E1 -22324.34,E2 -22324.34} C_VEL
LIN {X 0,Y 185.982,Z 265.312,A -85,B 0,C 180,E1 -22328.697,E2 -22328.697} C_VEL
LIN {X 0,Y 185.735,Z 265.349,A -85,B 0,C 180,E1 -22333.126,E2 -22333.126} C_VEL
LIN {X 0,Y 185.697,Z 265.349,A -85,B 0,C 180,E1 -22337.628,E2 -22337.628} C_VEL
LIN {X 0,Y 185.605,Z 265.364,A -85,B 0,C 180,E1 -22342.254,E2 -22342.254} C_VEL
LIN {X 0,Y 185.569,Z 265.371,A -85,B 0,C 180,E1 -22347.035,E2 -22347.035} C_VEL
LIN {X 0,Y 185.57,Z 265.37,A -85,B 0,C 180,E1 -22352.024,E2 -22352.024} C_VEL
LIN {X 0,Y 185.62,Z 265.544,A -85,B 0,C 180,E1 -22352.838,E2 -22352.838} C_VEL
LIN {X 0,Y 186.219,Z 269.049,A -85,B 0,C 180,E1 -22357.574,E2 -22357.574} C_VEL
LIN {X 0,Y 186.936,Z 273.046,A -85,B 0,C 180,E1 -22362.592,E2 -22362.592} C_VEL
LIN {X 0,Y 187.804,Z 277.305,A -85,B 0,C 180,E1 -22367.653,E2 -22367.653} C_VEL
LIN {X 0,Y 188.246,Z 279.938,A -85,B 0,C 180,E1 -22370.603,E2 -22370.603} C_VEL
LIN {X 0,Y 188.042,Z 282.459,A -85,B 0,C 180,E1 -22373.272,E2 -22373.272} C_VEL
LIN {X 0,Y 187.615,Z 284.224,A -85,B 0,C 180,E1 -22374.882,E2 -22374.882} C_VEL
LIN {X 0,Y 190.055,Z 297.723,A -85,B 0,C 180,E1 -22376.31,E2 -22376.31} C_VEL
LIN {X 0,Y 191.648,Z 310.57,A -85,B 0,C 180,E1 -22378.001,E2 -22378.001} C_VEL
LIN {X 0,Y 192.552,Z 322.083,A -85,B 0,C 180,E1 -22379.837,E2 -22379.837} C_VEL
LIN {X 0,Y 193.015,Z 332.139,A -85,B 0,C 180,E1 -22381.747,E2 -22381.747} C_VEL
LIN {X 0,Y 193.035,Z 342.672,A -85,B 0,C 180,E1 -22384.093,E2 -22384.093} C_VEL
LIN {X 0,Y 192.551,Z 345.946,A -85,B 0,C 180,E1 -22384.892,E2 -22384.892} C_VEL
LIN {X 0,Y 190.116,Z 355.693,A -85,B 0,C 180,E1 -22387.551,E2 -22387.551} C_VEL
LIN {X 0,Y 188.017,Z 363.817,A -85,B 0,C 180,E1 -22390.34,E2 -22390.34} C_VEL
LIN {X 0,Y 186.109,Z 371.272,A -85,B 0,C 180,E1 -22393.546,E2 -22393.546} C_VEL
LIN {X 0,Y 184.7,Z 377.251,A -85,B 0,C 180,E1 -22396.801,E2 -22396.801} C_VEL
LIN {X 0,Y 183.907,Z 381.972,A -85,B 0,C 180,E1 -22400.097,E2 -22400.097} C_VEL
LIN {X 0,Y 183.526,Z 385.547,A -85,B 0,C 180,E1 -22403.402,E2 -22403.402} C_VEL
LIN {X 0,Y 183.461,Z 387.365,A -85,B 0,C 180,E1 -22405.605,E2 -22405.605} C_VEL
LIN {X 0,Y 183.511,Z 388.701,A -85,B 0,C 180,E1 -22407.804,E2 -22407.804} C_VEL
LIN {X 0,Y 183.544,Z 389.614,A -85,B 0,C 180,E1 -22409.999,E2 -22409.999} C_VEL
LIN {X 0,Y 183.388,Z 390.132,A -85,B 0,C 180,E1 -22412.686,E2 -22412.686} C_VEL
LIN {X 0,Y 182.639,Z 390.159,A -85,B 0,C 180,E1 -22414.52,E2 -22414.52} C_VEL
LIN {X 0,Y 179.878,Z 389.485,A -85,B 0,C 180,E1 -22417.528,E2 -22417.528} C_VEL
LIN {X 0,Y 177.799,Z 388.547,A -85,B 0,C 180,E1 -22419.981,E2 -22419.981} C_VEL
LIN {X 0,Y 177.204,Z 387.589,A -85,B 0,C 180,E1 -22421.864,E2 -22421.864} C_VEL
LIN {X 0,Y 177.307,Z 387.169,A -85,B 0,C 180,E1 -22422.492,E2 -22422.492} C_VEL
LIN {X 0,Y 179.364,Z 383.531,A -85,B 0,C 180,E1 -22427.089,E2 -22427.089} C_VEL
LIN {X 0,Y 181.653,Z 379.707,A -85,B 0,C 180,E1 -22430.376,E2 -22430.376} C_VEL
LIN {X 0,Y 185.059,Z 373.937,A -85,B 0,C 180,E1 -22434.088,E2 -22434.088} C_VEL
LIN {X 0,Y 188.455,Z 367.699,A -85,B 0,C 180,E1 -22437.182,E2 -22437.182} C_VEL
LIN {X 0,Y 192.64,Z 360.091,A -85,B 0,C 180,E1 -22440.107,E2 -22440.107} C_VEL
LIN {X 0,Y 194.863,Z 355.66,A -85,B 0,C 180,E1 -22441.53,E2 -22441.53} C_VEL
LIN {X 0,Y 197.501,Z 347.421,A -85,B 0,C 180,E1 -22444.086,E2 -22444.086} C_VEL
LIN {X 0,Y 199.158,Z 339.051,A -85,B 0,C 180,E1 -22446.493,E2 -22446.493} C_VEL
LIN {X 0,Y 200.152,Z 329.178,A -85,B 0,C 180,E1 -22449.199,E2 -22449.199} C_VEL
LIN {X 0,Y 200.044,Z 319.481,A -85,B 0,C 180,E1 -22451.874,E2 -22451.874} C_VEL
LIN {X 0,Y 199.518,Z 314.588,A -85,B 0,C 180,E1 -22453.321,E2 -22453.321} C_VEL
LIN {X 0,Y 198.014,Z 309.433,A -85,B 0,C 180,E1 -22455.221,E2 -22455.221} C_VEL
LIN {X 0,Y 195.358,Z 302.537,A -85,B 0,C 180,E1 -22458.187,E2 -22458.187} C_VEL
LIN {X 0,Y 193.699,Z 299.241,A -85,B 0,C 180,E1 -22459.902,E2 -22459.902} C_VEL
LIN {X 0,Y 193.277,Z 297.942,A -85,B 0,C 180,E1 -22460.475,E2 -22460.475} C_VEL
LIN {X 0,Y 190.449,Z 292.632,A -85,B 0,C 180,E1 -22463.808,E2 -22463.808} C_VEL
LIN {X 0,Y 190.073,Z 291.43,A -85,B 0,C 180,E1 -22464.433,E2 -22464.433} C_VEL
LIN {X 0,Y 185.79,Z 283.164,A -85,B 0,C 180,E1 -22472.161,E2 -22472.161} C_VEL
LIN {X 0,Y 185.522,Z 282.486,A -85,B 0,C 180,E1 -22472.958,E2 -22472.958} C_VEL
LIN {X 0,Y 184.473,Z 280.638,A -85,B 0,C 180,E1 -22478.778,E2 -22478.778} C_VEL
LIN {X 0,Y 184.885,Z 280.168,A -85,B 0,C 180,E1 -22482.292,E2 -22482.292} C_VEL
LIN {X 0,Y 185.615,Z 280.535,A -85,B 0,C 180,E1 -22484.908,E2 -22484.908} C_VEL
LIN {X 0,Y 187.692,Z 283.35,A -85,B 0,C 180,E1 -22489.751,E2 -22489.751} C_VEL
LIN {X 0,Y 188.948,Z 284.17,A -85,B 0,C 180,E1 -22491.44,E2 -22491.44} C_VEL
LIN {X 0,Y 189.835,Z 285.294,A -85,B 0,C 180,E1 -22492.739,E2 -22492.739} C_VEL
LIN {X 0,Y 190.747,Z 287.108,A -85,B 0,C 180,E1 -22494.144,E2 -22494.144} C_VEL
LIN {X 0,Y 193.069,Z 289.453,A -85,B 0,C 180,E1 -22496.629,E2 -22496.629} C_VEL
LIN {X 0,Y 195.127,Z 293.028,A -85,B 0,C 180,E1 -22498.965,E2 -22498.965} C_VEL
LIN {X 0,Y 198.281,Z 299.755,A -85,B 0,C 180,E1 -22502.569,E2 -22502.569} C_VEL
LIN {X 0,Y 200.391,Z 305.015,A -85,B 0,C 180,E1 -22505.027,E2 -22505.027} C_VEL
LIN {X 0,Y 202.096,Z 311.569,A -85,B 0,C 180,E1 -22507.614,E2 -22507.614} C_VEL
LIN {X 0,Y 203.133,Z 319.445,A -85,B 0,C 180,E1 -22510.462,E2 -22510.462} C_VEL
LIN {X 0,Y 203.15,Z 327.201,A -85,B 0,C 180,E1 -22513.14,E2 -22513.14} C_VEL
LIN {X 0,Y 201.731,Z 330.931,A -85,B 0,C 180,E1 -22514.111,E2 -22514.111} C_VEL
LIN {X 0,Y 197.52,Z 339.549,A -85,B 0,C 180,E1 -22516.534,E2 -22516.534} C_VEL
LIN {X 0,Y 193.5,Z 347.025,A -85,B 0,C 180,E1 -22519.212,E2 -22519.212} C_VEL
LIN {X 0,Y 189.655,Z 353.404,A -85,B 0,C 180,E1 -22522.121,E2 -22522.121} C_VEL
LIN {X 0,Y 186.318,Z 358.521,A -85,B 0,C 180,E1 -22525.141,E2 -22525.141} C_VEL
LIN {X 0,Y 183.537,Z 362.545,A -85,B 0,C 180,E1 -22528.274,E2 -22528.274} C_VEL
LIN {X 0,Y 181.18,Z 365.562,A -85,B 0,C 180,E1 -22531.421,E2 -22531.421} C_VEL
LIN {X 0,Y 179.343,Z 367.664,A -85,B 0,C 180,E1 -22534.623,E2 -22534.623} C_VEL
LIN {X 0,Y 177.406,Z 369.184,A -85,B 0,C 180,E1 -22539.329,E2 -22539.329} C_VEL
LIN {X 0,Y 176.588,Z 369.256,A -85,B 0,C 180,E1 -22542.571,E2 -22542.571} C_VEL
LIN {X 0,Y 176.101,Z 367.96,A -85,B 0,C 180,E1 -22547.279,E2 -22547.279} C_VEL
LIN {X 0,Y 176.21,Z 366.171,A -85,B 0,C 180,E1 -22550.348,E2 -22550.348} C_VEL
LIN {X 0,Y 176.696,Z 363.678,A -85,B 0,C 180,E1 -22553.374,E2 -22553.374} C_VEL
LIN {X 0,Y 177.438,Z 360.483,A -85,B 0,C 180,E1 -22556.324,E2 -22556.324} C_VEL
LIN {X 0,Y 178.644,Z 355.374,A -85,B 0,C 180,E1 -22559.931,E2 -22559.931} C_VEL
LIN {X 0,Y 180.394,Z 348.547,A -85,B 0,C 180,E1 -22563.635,E2 -22563.635} C_VEL
LIN {X 0,Y 182.343,Z 341.317,A -85,B 0,C 180,E1 -22566.733,E2 -22566.733} C_VEL
LIN {X 0,Y 184.893,Z 331.674,A -85,B 0,C 180,E1 -22569.996,E2 -22569.996} C_VEL
LIN {X 0,Y 187.544,Z 320.968,A -85,B 0,C 180,E1 -22572.838,E2 -22572.838} C_VEL
LIN {X 0,Y 189.81,Z 310.774,A -85,B 0,C 180,E1 -22574.98,E2 -22574.98} C_VEL
LIN {X 0,Y 188.15,Z 299.67,A -85,B 0,C 180,E1 -22577.325,E2 -22577.325} C_VEL
LIN {X 0,Y 185.578,Z 287.767,A -85,B 0,C 180,E1 -22579.533,E2 -22579.533} C_VEL
LIN {X 0,Y 182.185,Z 275.643,A -85,B 0,C 180,E1 -22581.509,E2 -22581.509} C_VEL
LIN {X 0,Y 178.762,Z 266.658,A -85,B 0,C 180,E1 -22582.873,E2 -22582.873} C_VEL
LIN {X 0,Y 178.717,Z 266.225,A -85,B 0,C 180,E1 -22582.942,E2 -22582.942} C_VEL
LIN {X 0,Y 179.13,Z 266.176,A -85,B 0,C 180,E1 -22587.753,E2 -22587.753} C_VEL
LIN {X 0,Y 179.358,Z 266.146,A -85,B 0,C 180,E1 -22590.001,E2 -22590.001} C_VEL
LIN {X 0,Y 178.862,Z 266.205,A -85,B 0,C 180,E1 -22594.508,E2 -22594.508} C_VEL
LIN {X 0,Y 178.947,Z 266.196,A -85,B 0,C 180,E1 -22599.04,E2 -22599.04} C_VEL
LIN {X 0,Y 178.678,Z 266.231,A -85,B 0,C 180,E1 -22603.652,E2 -22603.652} C_VEL
LIN {X 0,Y 178.67,Z 266.227,A -85,B 0,C 180,E1 -22608.343,E2 -22608.343} C_VEL
LIN {X 0,Y 178.524,Z 266.251,A -85,B 0,C 180,E1 -22613.184,E2 -22613.184} C_VEL
LIN {X 0,Y 178.478,Z 266.249,A -85,B 0,C 180,E1 -22618.2,E2 -22618.2} C_VEL
LIN {X 0,Y 178.491,Z 266.255,A -85,B 0,C 180,E1 -22620.79,E2 -22620.79} C_VEL
LIN {X 0,Y 178.476,Z 266.251,A -85,B 0,C 180,E1 -22624.223,E2 -22624.223} C_VEL
LIN {X 0,Y 178.479,Z 266.251,A -85,B 0,C 180,E1 -22629.054,E2 -22629.054} C_VEL
LIN {X 0,Y 178.51,Z 266.249,A -85,B 0,C 180,E1 -22632.014,E2 -22632.014} C_VEL
LIN {X 0,Y 178.523,Z 266.24,A -85,B 0,C 180,E1 -22635.124,E2 -22635.124} C_VEL
LIN {X 0,Y 178.511,Z 266.234,A -85,B 0,C 180,E1 -22638.422,E2 -22638.422} C_VEL
LIN {X 0,Y 178.483,Z 266.252,A -85,B 0,C 180,E1 -22643.803,E2 -22643.803} C_VEL
LIN {X 0,Y 178.488,Z 266.246,A -85,B 0,C 180,E1 -22646.552,E2 -22646.552} C_VEL
LIN {X 0,Y 178.52,Z 266.231,A -85,B 0,C 180,E1 -22650.01,E2 -22650.01} C_VEL
LIN {X 0,Y 178.533,Z 266.244,A -85,B 0,C 180,E1 -22654.88,E2 -22654.88} C_VEL
LIN {X 0,Y 178.623,Z 266.223,A -85,B 0,C 180,E1 -22660.788,E2 -22660.788} C_VEL
LIN {X 0,Y 178.659,Z 266.227,A -85,B 0,C 180,E1 -22666.352,E2 -22666.352} C_VEL
LIN {X 0,Y 178.912,Z 266.196,A -85,B 0,C 180,E1 -22670.964,E2 -22670.964} C_VEL
LIN {X 0,Y 179.154,Z 266.161,A -85,B 0,C 180,E1 -22677.756,E2 -22677.756} C_VEL
LIN {X 0,Y 179.373,Z 266.142,A -85,B 0,C 180,E1 -22680.004,E2 -22680.004} C_VEL
LIN {X 0,Y 178.863,Z 266.199,A -85,B 0,C 180,E1 -22684.511,E2 -22684.511} C_VEL
LIN {X 0,Y 178.912,Z 266.193,A -85,B 0,C 180,E1 -22689.044,E2 -22689.044} C_VEL
LIN {X 0,Y 178.663,Z 266.228,A -85,B 0,C 180,E1 -22693.655,E2 -22693.655} C_VEL
LIN {X 0,Y 178.631,Z 266.233,A -85,B 0,C 180,E1 -22699.219,E2 -22699.219} C_VEL
LIN {X 0,Y 178.543,Z 266.246,A -85,B 0,C 180,E1 -22705.127,E2 -22705.127} C_VEL
LIN {X 0,Y 178.516,Z 266.249,A -85,B 0,C 180,E1 -22710.788,E2 -22710.788} C_VEL
LIN {X 0,Y 178.531,Z 266.29,A -85,B 0,C 180,E1 -22712.107,E2 -22712.107} C_VEL
LIN {X 0,Y 178.99,Z 269.101,A -85,B 0,C 180,E1 -22716.088,E2 -22716.088} C_VEL
LIN {X 0,Y 179.538,Z 272.203,A -85,B 0,C 180,E1 -22720.237,E2 -22720.237} C_VEL
LIN {X 0,Y 180.358,Z 276.334,A -85,B 0,C 180,E1 -22725.459,E2 -22725.459} C_VEL
LIN {X 0,Y 180.933,Z 279.022,A -85,B 0,C 180,E1 -22728.673,E2 -22728.673} C_VEL
LIN {X 0,Y 181.156,Z 281.619,A -85,B 0,C 180,E1 -22731.63,E2 -22731.63} C_VEL
LIN {X 0,Y 180.793,Z 283.798,A -85,B 0,C 180,E1 -22733.808,E2 -22733.808} C_VEL
LIN {X 0,Y 183.165,Z 296.762,A -85,B 0,C 180,E1 -22735.255,E2 -22735.255} C_VEL
LIN {X 0,Y 184.681,Z 308.528,A -85,B 0,C 180,E1 -22736.851,E2 -22736.851} C_VEL
LIN {X 0,Y 185.668,Z 320.917,A -85,B 0,C 180,E1 -22738.873,E2 -22738.873} C_VEL
LIN {X 0,Y 186.168,Z 332.896,A -85,B 0,C 180,E1 -22741.227,E2 -22741.227} C_VEL
LIN {X 0,Y 186.099,Z 343.217,A -85,B 0,C 180,E1 -22743.656,E2 -22743.656} C_VEL
LIN {X 0,Y 185.272,Z 347.457,A -85,B 0,C 180,E1 -22744.737,E2 -22744.737} C_VEL
LIN {X 0,Y 182.911,Z 356.492,A -85,B 0,C 180,E1 -22747.403,E2 -22747.403} C_VEL
LIN {X 0,Y 180.533,Z 365.321,A -85,B 0,C 180,E1 -22750.676,E2 -22750.676} C_VEL
LIN {X 0,Y 178.697,Z 372.415,A -85,B 0,C 180,E1 -22754.019,E2 -22754.019} C_VEL
LIN {X 0,Y 177.402,Z 378.057,A -85,B 0,C 180,E1 -22757.414,E2 -22757.414} C_VEL
LIN {X 0,Y 176.685,Z 382.484,A -85,B 0,C 180,E1 -22760.844,E2 -22760.844} C_VEL
LIN {X 0,Y 176.436,Z 386.2,A -85,B 0,C 180,E1 -22764.798,E2 -22764.798} C_VEL
LIN {X 0,Y 176.449,Z 388.101,A -85,B 0,C 180,E1 -22767.716,E2 -22767.716} C_VEL
LIN {X 0,Y 176.48,Z 389.06,A -85,B 0,C 180,E1 -22769.999,E2 -22769.999} C_VEL
LIN {X 0,Y 176.315,Z 389.625,A -85,B 0,C 180,E1 -22772.635,E2 -22772.635} C_VEL
LIN {X 0,Y 176.305,Z 389.511,A -85,B 0,C 180,E1 -22776.867,E2 -22776.867} C_VEL
LIN {X 0,Y 177.012,Z 387.816,A -85,B 0,C 180,E1 -22781.449,E2 -22781.449} C_VEL
LIN {X 0,Y 177.307,Z 387.169,A -85,B 0,C 180,E1 -22782.492,E2 -22782.492} C_VEL
LIN {X 0,Y 177.321,Z 385.98,A -85,B 0,C 180,E1 -22784.36,E2 -22784.36} C_VEL
LIN {X 0,Y 175.976,Z 383.473,A -85,B 0,C 180,E1 -22787.448,E2 -22787.448} C_VEL
LIN {X 0,Y 175.142,Z 381.12,A -85,B 0,C 180,E1 -22789.909,E2 -22789.909} C_VEL
LIN {X 0,Y 175.504,Z 379.053,A -85,B 0,C 180,E1 -22791.717,E2 -22791.717} C_VEL
LIN {X 0,Y 175.922,Z 378.298,A -85,B 0,C 180,E1 -22792.297,E2 -22792.297} C_VEL
LIN {X 0,Y 179.128,Z 373.214,A -85,B 0,C 180,E1 -22795.566,E2 -22795.566} C_VEL
LIN {X 0,Y 182.877,Z 366.969,A -85,B 0,C 180,E1 -22798.708,E2 -22798.708} C_VEL
LIN {X 0,Y 187.389,Z 359.295,A -85,B 0,C 180,E1 -22801.671,E2 -22801.671} C_VEL
LIN {X 0,Y 189.444,Z 354.872,A -85,B 0,C 180,E1 -22803.173,E2 -22803.173} C_VEL
LIN {X 0,Y 192.117,Z 346.64,A -85,B 0,C 180,E1 -22805.823,E2 -22805.823} C_VEL
LIN {X 0,Y 193.921,Z 337.903,A -85,B 0,C 180,E1 -22808.471,E2 -22808.471} C_VEL
LIN {X 0,Y 194.807,Z 329.627,A -85,B 0,C 180,E1 -22810.891,E2 -22810.891} C_VEL
LIN {X 0,Y 194.897,Z 321.759,A -85,B 0,C 180,E1 -22813.245,E2 -22813.245} C_VEL
LIN {X 0,Y 194.406,Z 317.496,A -85,B 0,C 180,E1 -22814.69,E2 -22814.69} C_VEL
LIN {X 0,Y 193.007,Z 312.58,A -85,B 0,C 180,E1 -22816.739,E2 -22816.739} C_VEL
LIN {X 0,Y 191.6,Z 308.426,A -85,B 0,C 180,E1 -22818.677,E2 -22818.677} C_VEL
LIN {X 0,Y 189.012,Z 302.132,A -85,B 0,C 180,E1 -22822.151,E2 -22822.151} C_VEL
LIN {X 0,Y 186.507,Z 296.483,A -85,B 0,C 180,E1 -22825.994,E2 -22825.994} C_VEL
LIN {X 0,Y 183.575,Z 289.748,A -85,B 0,C 180,E1 -22832.647,E2 -22832.647} C_VEL
LIN {X 0,Y 182.982,Z 288.543,A -85,B 0,C 180,E1 -22835.004,E2 -22835.004} C_VEL
LIN {X 0,Y 182.591,Z 287.308,A -85,B 0,C 180,E1 -22839.728,E2 -22839.728} C_VEL
LIN {X 0,Y 183.222,Z 287.081,A -85,B 0,C 180,E1 -22843.52,E2 -22843.52} C_VEL
LIN {X 0,Y 183.49,Z 287.148,A -85,B 0,C 180,E1 -22844.444,E2 -22844.444} C_VEL
LIN {X 0,Y 185.566,Z 290.205,A -85,B 0,C 180,E1 -22849.958,E2 -22849.958} C_VEL
LIN {X 0,Y 186.486,Z 290.864,A -85,B 0,C 180,E1 -22851.326,E2 -22851.326} C_VEL
LIN {X 0,Y 188.55,Z 294.278,A -85,B 0,C 180,E1 -22854.65,E2 -22854.65} C_VEL
LIN {X 0,Y 190.087,Z 296.308,A -85,B 0,C 180,E1 -22856.594,E2 -22856.594} C_VEL
LIN {X 0,Y 192.081,Z 300.395,A -85,B 0,C 180,E1 -22859.307,E2 -22859.307} C_VEL
LIN {X 0,Y 194.663,Z 306.424,A -85,B 0,C 180,E1 -22862.721,E2 -22862.721} C_VEL
LIN {X 0,Y 196.296,Z 312.191,A -85,B 0,C 180,E1 -22865.389,E2 -22865.389} C_VEL
LIN {X 0,Y 197.226,Z 317.869,A -85,B 0,C 180,E1 -22867.726,E2 -22867.726} C_VEL
LIN {X 0,Y 197.6,Z 324.44,A -85,B 0,C 180,E1 -22870.24,E2 -22870.24} C_VEL
LIN {X 0,Y 197.161,Z 330.195,A -85,B 0,C 180,E1 -22872.346,E2 -22872.346} C_VEL
LIN {X 0,Y 192.78,Z 338.944,A -85,B 0,C 180,E1 -22874.781,E2 -22874.781} C_VEL
LIN {X 0,Y 187.996,Z 347.36,A -85,B 0,C 180,E1 -22877.79,E2 -22877.79} C_VEL
LIN {X 0,Y 183.444,Z 354.368,A -85,B 0,C 180,E1 -22881.101,E2 -22881.101} C_VEL
LIN {X 0,Y 180.096,Z 359.163,A -85,B 0,C 180,E1 -22884.048,E2 -22884.048} C_VEL
LIN {X 0,Y 177.267,Z 362.962,A -85,B 0,C 180,E1 -22887.094,E2 -22887.094} C_VEL
LIN {X 0,Y 174.859,Z 365.839,A -85,B 0,C 180,E1 -22890.154,E2 -22890.154} C_VEL
LIN {X 0,Y 173.729,Z 367.049,A -85,B 0,C 180,E1 -22891.842,E2 -22891.842} C_VEL
LIN {X 0,Y 171.92,Z 368.738,A -85,B 0,C 180,E1 -22895.159,E2 -22895.159} C_VEL
LIN {X 0,Y 170.582,Z 369.621,A -85,B 0,C 180,E1 -22898.485,E2 -22898.485} C_VEL
LIN {X 0,Y 169.644,Z 369.741,A -85,B 0,C 180,E1 -22901.783,E2 -22901.783} C_VEL
LIN {X 0,Y 169.133,Z 369.106,A -85,B 0,C 180,E1 -22905.059,E2 -22905.059} C_VEL
LIN {X 0,Y 169.011,Z 367.634,A -85,B 0,C 180,E1 -22908.453,E2 -22908.453} C_VEL
LIN {X 0,Y 169.33,Z 365.184,A -85,B 0,C 180,E1 -22912.047,E2 -22912.047} C_VEL
LIN {X 0,Y 170.12,Z 361.653,A -85,B 0,C 180,E1 -22915.706,E2 -22915.706} C_VEL
LIN {X 0,Y 171.3,Z 356.773,A -85,B 0,C 180,E1 -22919.485,E2 -22919.485} C_VEL
LIN {X 0,Y 173.028,Z 350.282,A -85,B 0,C 180,E1 -22923.317,E2 -22923.317} C_VEL
LIN {X 0,Y 175.144,Z 342.67,A -85,B 0,C 180,E1 -22926.81,E2 -22926.81} C_VEL
LIN {X 0,Y 177.625,Z 333.667,A -85,B 0,C 180,E1 -22930.085,E2 -22930.085} C_VEL
LIN {X 0,Y 180.343,Z 323.382,A -85,B 0,C 180,E1 -22933.007,E2 -22933.007} C_VEL
LIN {X 0,Y 183.018,Z 311.922,A -85,B 0,C 180,E1 -22935.578,E2 -22935.578} C_VEL
LIN {X 0,Y 181.482,Z 301.144,A -85,B 0,C 180,E1 -22937.987,E2 -22937.987} C_VEL
LIN {X 0,Y 179.241,Z 290.361,A -85,B 0,C 180,E1 -22940.124,E2 -22940.124} C_VEL
LIN {X 0,Y 176.431,Z 279.704,A -85,B 0,C 180,E1 -22941.986,E2 -22941.986} C_VEL
LIN {X 0,Y 172.767,Z 270.047,A -85,B 0,C 180,E1 -22943.615,E2 -22943.615} C_VEL
LIN {X 0,Y 171.695,Z 267.102,A -85,B 0,C 180,E1 -22944.128,E2 -22944.128} C_VEL
LIN {X 0,Y 172.074,Z 267.055,A -85,B 0,C 180,E1 -22947.661,E2 -22947.661} C_VEL
LIN {X 0,Y 172.32,Z 267.023,A -85,B 0,C 180,E1 -22950.001,E2 -22950.001} C_VEL
LIN {X 0,Y 171.811,Z 267.084,A -85,B 0,C 180,E1 -22954.694,E2 -22954.694} C_VEL
LIN {X 0,Y 171.876,Z 267.077,A -85,B 0,C 180,E1 -22959.415,E2 -22959.415} C_VEL
LIN {X 0,Y 171.603,Z 267.112,A -85,B 0,C 180,E1 -22964.226,E2 -22964.226} C_VEL
LIN {X 0,Y 171.566,Z 267.114,A -85,B 0,C 180,E1 -22969.595,E2 -22969.595} C_VEL
LIN {X 0,Y 171.466,Z 267.123,A -85,B 0,C 180,E1 -22975.625,E2 -22975.625} C_VEL
LIN {X 0,Y 171.449,Z 267.131,A -85,B 0,C 180,E1 -22980.599,E2 -22980.599} C_VEL
LIN {X 0,Y 171.399,Z 267.126,A -85,B 0,C 180,E1 -22985.035,E2 -22985.035} C_VEL
LIN {X 0,Y 171.431,Z 267.127,A -85,B 0,C 180,E1 -22988.845,E2 -22988.845} C_VEL
LIN {X 0,Y 171.447,Z 267.126,A -85,B 0,C 180,E1 -22994.178,E2 -22994.178} C_VEL
LIN {X 0,Y 171.428,Z 267.121,A -85,B 0,C 180,E1 -22999.014,E2 -22999.014} C_VEL
LIN {X 0,Y 171.439,Z 267.128,A -85,B 0,C 180,E1 -23002.06,E2 -23002.06} C_VEL
LIN {X 0,Y 171.412,Z 267.13,A -85,B 0,C 180,E1 -23005.088,E2 -23005.088} C_VEL
LIN {X 0,Y 171.446,Z 267.112,A -85,B 0,C 180,E1 -23010.539,E2 -23010.539} C_VEL
LIN {X 0,Y 171.456,Z 267.127,A -85,B 0,C 180,E1 -23015.806,E2 -23015.806} C_VEL
LIN {X 0,Y 171.579,Z 267.1,A -85,B 0,C 180,E1 -23020.876,E2 -23020.876} C_VEL
LIN {X 0,Y 171.576,Z 267.105,A -85,B 0,C 180,E1 -23025.777,E2 -23025.777} C_VEL
LIN {X 0,Y 171.849,Z 267.077,A -85,B 0,C 180,E1 -23030.589,E2 -23030.589} C_VEL
LIN {X 0,Y 171.815,Z 267.066,A -85,B 0,C 180,E1 -23035.311,E2 -23035.311} C_VEL
LIN {X 0,Y 172.336,Z 267.018,A -85,B 0,C 180,E1 -23040.004,E2 -23040.004} C_VEL
LIN {X 0,Y 171.812,Z 267.077,A -85,B 0,C 180,E1 -23044.697,E2 -23044.697} C_VEL
LIN {X 0,Y 171.85,Z 267.074,A -85,B 0,C 180,E1 -23049.419,E2 -23049.419} C_VEL
LIN {X 0,Y 171.581,Z 267.107,A -85,B 0,C 180,E1 -23054.231,E2 -23054.231} C_VEL
LIN {X 0,Y 171.552,Z 267.117,A -85,B 0,C 180,E1 -23059.565,E2 -23059.565} C_VEL
LIN {X 0,Y 171.477,Z 267.126,A -85,B 0,C 180,E1 -23065.619,E2 -23065.619} C_VEL
LIN {X 0,Y 171.464,Z 267.158,A -85,B 0,C 180,E1 -23071.518,E2 -23071.518} C_VEL
LIN {X 0,Y 171.885,Z 269.6,A -85,B 0,C 180,E1 -23075.137,E2 -23075.137} C_VEL
LIN {X 0,Y 172.584,Z 273.555,A -85,B 0,C 180,E1 -23080.663,E2 -23080.663} C_VEL
LIN {X 0,Y 173.263,Z 276.893,A -85,B 0,C 180,E1 -23085.05,E2 -23085.05} C_VEL
LIN {X 0,Y 173.982,Z 280.69,A -85,B 0,C 180,E1 -23089.734,E2 -23089.734} C_VEL
LIN {X 0,Y 173.971,Z 282.909,A -85,B 0,C 180,E1 -23092.336,E2 -23092.336} C_VEL
LIN {X 0,Y 173.95,Z 283.183,A -85,B 0,C 180,E1 -23092.65,E2 -23092.65} C_VEL
LIN {X 0,Y 176.263,Z 295.528,A -85,B 0,C 180,E1 -23094.089,E2 -23094.089} C_VEL
LIN {X 0,Y 177.843,Z 307.054,A -85,B 0,C 180,E1 -23095.709,E2 -23095.709} C_VEL
LIN {X 0,Y 178.748,Z 318.497,A -85,B 0,C 180,E1 -23097.607,E2 -23097.607} C_VEL
LIN {X 0,Y 179.292,Z 331.022,A -85,B 0,C 180,E1 -23100.121,E2 -23100.121} C_VEL
LIN {X 0,Y 179.239,Z 341.268,A -85,B 0,C 180,E1 -23102.565,E2 -23102.565} C_VEL
LIN {X 0,Y 178.85,Z 345.765,A -85,B 0,C 180,E1 -23103.762,E2 -23103.762} C_VEL
LIN {X 0,Y 176.352,Z 355.06,A -85,B 0,C 180,E1 -23106.513,E2 -23106.513} C_VEL
LIN {X 0,Y 173.818,Z 364.053,A -85,B 0,C 180,E1 -23109.897,E2 -23109.897} C_VEL
LIN {X 0,Y 171.847,Z 371.307,A -85,B 0,C 180,E1 -23113.363,E2 -23113.363} C_VEL
LIN {X 0,Y 170.462,Z 377.112,A -85,B 0,C 180,E1 -23116.892,E2 -23116.892} C_VEL
LIN {X 0,Y 169.659,Z 381.66,A -85,B 0,C 180,E1 -23120.461,E2 -23120.461} C_VEL
LIN {X 0,Y 169.365,Z 385.689,A -85,B 0,C 180,E1 -23124.849,E2 -23124.849} C_VEL
LIN {X 0,Y 169.387,Z 387.47,A -85,B 0,C 180,E1 -23127.621,E2 -23127.621} C_VEL
LIN {X 0,Y 169.416,Z 388.505,A -85,B 0,C 180,E1 -23129.999,E2 -23129.999} C_VEL
LIN {X 0,Y 169.185,Z 389.286,A -85,B 0,C 180,E1 -23134.423,E2 -23134.423} C_VEL
LIN {X 0,Y 169.243,Z 389.104,A -85,B 0,C 180,E1 -23137.155,E2 -23137.155} C_VEL
LIN {X 0,Y 169.51,Z 388.539,A -85,B 0,C 180,E1 -23139.545,E2 -23139.545} C_VEL
LIN {X 0,Y 170.792,Z 386.21,A -85,B 0,C 180,E1 -23144.293,E2 -23144.293} C_VEL
LIN {X 0,Y 172.576,Z 383.453,A -85,B 0,C 180,E1 -23147.783,E2 -23147.783} C_VEL
LIN {X 0,Y 174.979,Z 379.749,A -85,B 0,C 180,E1 -23151.19,E2 -23151.19} C_VEL
LIN {X 0,Y 175.922,Z 378.298,A -85,B 0,C 180,E1 -23152.297,E2 -23152.297} C_VEL
LIN {X 0,Y 176.852,Z 375.984,A -85,B 0,C 180,E1 -23154.037,E2 -23154.037} C_VEL
LIN {X 0,Y 176.943,Z 371.867,A -85,B 0,C 180,E1 -23156.96,E2 -23156.96} C_VEL
LIN {X 0,Y 177.401,Z 367.19,A -85,B 0,C 180,E1 -23159.777,E2 -23159.777} C_VEL
LIN {X 0,Y 178.855,Z 363.965,A -85,B 0,C 180,E1 -23161.297,E2 -23161.297} C_VEL
LIN {X 0,Y 182.91,Z 357.103,A -85,B 0,C 180,E1 -23163.856,E2 -23163.856} C_VEL
LIN {X 0,Y 185.896,Z 349.407,A -85,B 0,C 180,E1 -23166.543,E2 -23166.543} C_VEL
LIN {X 0,Y 188.155,Z 340.558,A -85,B 0,C 180,E1 -23169.417,E2 -23169.417} C_VEL
LIN {X 0,Y 189.484,Z 331.423,A -85,B 0,C 180,E1 -23172.308,E2 -23172.308} C_VEL
LIN {X 0,Y 189.824,Z 324.052,A -85,B 0,C 180,E1 -23174.703,E2 -23174.703} C_VEL
LIN {X 0,Y 189.022,Z 319.301,A -85,B 0,C 180,E1 -23176.66,E2 -23176.66} C_VEL
LIN {X 0,Y 187.264,Z 313.241,A -85,B 0,C 180,E1 -23179.65,E2 -23179.65} C_VEL
LIN {X 0,Y 185.429,Z 307.955,A -85,B 0,C 180,E1 -23182.74,E2 -23182.74} C_VEL
LIN {X 0,Y 183.591,Z 302.983,A -85,B 0,C 180,E1 -23186.21,E2 -23186.21} C_VEL
LIN {X 0,Y 181.009,Z 296.179,A -85,B 0,C 180,E1 -23193.252,E2 -23193.252} C_VEL
LIN {X 0,Y 180.293,Z 294.649,A -85,B 0,C 180,E1 -23197.054,E2 -23197.054} C_VEL
LIN {X 0,Y 180.511,Z 293.761,A -85,B 0,C 180,E1 -23201.848,E2 -23201.848} C_VEL
LIN {X 0,Y 181.077,Z 293.822,A -85,B 0,C 180,E1 -23204.232,E2 -23204.232} C_VEL
LIN {X 0,Y 183.666,Z 297.43,A -85,B 0,C 180,E1 -23211.192,E2 -23211.192} C_VEL
LIN {X 0,Y 186.267,Z 301.724,A -85,B 0,C 180,E1 -23215.669,E2 -23215.669} C_VEL
LIN {X 0,Y 188.011,Z 305.714,A -85,B 0,C 180,E1 -23218.587,E2 -23218.587} C_VEL
LIN {X 0,Y 190.159,Z 311.53,A -85,B 0,C 180,E1 -23222.114,E2 -23222.114} C_VEL
LIN {X 0,Y 191.38,Z 316.816,A -85,B 0,C 180,E1 -23224.736,E2 -23224.736} C_VEL
LIN {X 0,Y 191.971,Z 322.719,A -85,B 0,C 180,E1 -23227.358,E2 -23227.358} C_VEL
LIN {X 0,Y 191.895,Z 329.125,A -85,B 0,C 180,E1 -23229.961,E2 -23229.961} C_VEL
LIN {X 0,Y 191.56,Z 331.968,A -85,B 0,C 180,E1 -23231.102,E2 -23231.102} C_VEL
LIN {X 0,Y 187.014,Z 340.506,A -85,B 0,C 180,E1 -23233.619,E2 -23233.619} C_VEL
LIN {X 0,Y 182.338,Z 348.151,A -85,B 0,C 180,E1 -23236.46,E2 -23236.46} C_VEL
LIN {X 0,Y 177.376,Z 355.332,A -85,B 0,C 180,E1 -23239.974,E2 -23239.974} C_VEL
LIN {X 0,Y 173.803,Z 360.031,A -85,B 0,C 180,E1 -23243.024,E2 -23243.024} C_VEL
LIN {X 0,Y 170.021,Z 364.597,A -85,B 0,C 180,E1 -23247.041,E2 -23247.041} C_VEL
LIN {X 0,Y 167.594,Z 367.124,A -85,B 0,C 180,E1 -23250.208,E2 -23250.208} C_VEL
LIN {X 0,Y 165.598,Z 368.91,A -85,B 0,C 180,E1 -23253.48,E2 -23253.48} C_VEL
LIN {X 0,Y 164.041,Z 369.968,A -85,B 0,C 180,E1 -23256.85,E2 -23256.85} C_VEL
LIN {X 0,Y 162.897,Z 370.243,A -85,B 0,C 180,E1 -23260.322,E2 -23260.322} C_VEL
LIN {X 0,Y 162.15,Z 369.726,A -85,B 0,C 180,E1 -23263.9,E2 -23263.9} C_VEL
LIN {X 0,Y 161.9,Z 368.366,A -85,B 0,C 180,E1 -23267.551,E2 -23267.551} C_VEL
LIN {X 0,Y 162.33,Z 364.977,A -85,B 0,C 180,E1 -23272.692,E2 -23272.692} C_VEL
LIN {X 0,Y 163.075,Z 361.833,A -85,B 0,C 180,E1 -23275.928,E2 -23275.928} C_VEL
LIN {X 0,Y 164.598,Z 355.783,A -85,B 0,C 180,E1 -23280.594,E2 -23280.594} C_VEL
LIN {X 0,Y 166.521,Z 348.923,A -85,B 0,C 180,E1 -23284.566,E2 -23284.566} C_VEL
LIN {X 0,Y 168.696,Z 341.422,A -85,B 0,C 180,E1 -23287.981,E2 -23287.981} C_VEL
LIN {X 0,Y 170.998,Z 333.275,A -85,B 0,C 180,E1 -23290.947,E2 -23290.947} C_VEL
LIN {X 0,Y 173.76,Z 323.127,A -85,B 0,C 180,E1 -23293.89,E2 -23293.89} C_VEL
LIN {X 0,Y 176.187,Z 313.347,A -85,B 0,C 180,E1 -23296.154,E2 -23296.154} C_VEL
LIN {X 0,Y 175.025,Z 303.765,A -85,B 0,C 180,E1 -23298.419,E2 -23298.419} C_VEL
LIN {X 0,Y 172.983,Z 293.267,A -85,B 0,C 180,E1 -23300.649,E2 -23300.649} C_VEL
LIN {X 0,Y 169.945,Z 281.5,A -85,B 0,C 180,E1 -23302.875,E2 -23302.875} C_VEL
LIN {X 0,Y 166.616,Z 272.857,A -85,B 0,C 180,E1 -23304.48,E2 -23304.48} C_VEL
LIN {X 0,Y 164.882,Z 268.947,A -85,B 0,C 180,E1 -23305.188,E2 -23305.188} C_VEL
LIN {X 0,Y 164.722,Z 267.97,A -85,B 0,C 180,E1 -23305.413,E2 -23305.413} C_VEL
LIN {X 0,Y 165.282,Z 267.9,A -85,B 0,C 180,E1 -23310.001,E2 -23310.001} C_VEL
LIN {X 0,Y 164.761,Z 267.963,A -85,B 0,C 180,E1 -23314.895,E2 -23314.895} C_VEL
LIN {X 0,Y 164.839,Z 267.949,A -85,B 0,C 180,E1 -23317.35,E2 -23317.35} C_VEL
LIN {X 0,Y 164.741,Z 267.961,A -85,B 0,C 180,E1 -23321.154,E2 -23321.154} C_VEL
LIN {X 0,Y 164.517,Z 267.991,A -85,B 0,C 180,E1 -23327.401,E2 -23327.401} C_VEL
LIN {X 0,Y 164.509,Z 267.993,A -85,B 0,C 180,E1 -23329.986,E2 -23329.986} C_VEL
LIN {X 0,Y 164.389,Z 268.003,A -85,B 0,C 180,E1 -23336.141,E2 -23336.141} C_VEL
LIN {X 0,Y 164.379,Z 268.012,A -85,B 0,C 180,E1 -23341.239,E2 -23341.239} C_VEL
LIN {X 0,Y 164.343,Z 268.001,A -85,B 0,C 180,E1 -23346.778,E2 -23346.778} C_VEL
LIN {X 0,Y 164.368,Z 268.008,A -85,B 0,C 180,E1 -23349.895,E2 -23349.895} C_VEL
LIN {X 0,Y 164.385,Z 268.006,A -85,B 0,C 180,E1 -23353.388,E2 -23353.388} C_VEL
LIN {X 0,Y 164.389,Z 267.99,A -85,B 0,C 180,E1 -23356.847,E2 -23356.847} C_VEL
LIN {X 0,Y 164.371,Z 268.003,A -85,B 0,C 180,E1 -23360.322,E2 -23360.322} C_VEL
LIN {X 0,Y 164.365,Z 268.011,A -85,B 0,C 180,E1 -23364.334,E2 -23364.334} C_VEL
LIN {X 0,Y 164.388,Z 267.991,A -85,B 0,C 180,E1 -23369.139,E2 -23369.139} C_VEL
LIN {X 0,Y 164.415,Z 268.003,A -85,B 0,C 180,E1 -23374.699,E2 -23374.699} C_VEL
LIN {X 0,Y 164.484,Z 267.987,A -85,B 0,C 180,E1 -23380.056,E2 -23380.056} C_VEL
LIN {X 0,Y 164.524,Z 267.982,A -85,B 0,C 180,E1 -23385.154,E2 -23385.154} C_VEL
LIN {X 0,Y 164.769,Z 267.96,A -85,B 0,C 180,E1 -23390.181,E2 -23390.181} C_VEL
LIN {X 0,Y 164.831,Z 267.945,A -85,B 0,C 180,E1 -23392.655,E2 -23392.655} C_VEL
LIN {X 0,Y 165.05,Z 267.915,A -85,B 0,C 180,E1 -23397.564,E2 -23397.564} C_VEL
LIN {X 0,Y 165.298,Z 267.895,A -85,B 0,C 180,E1 -23400.004,E2 -23400.004} C_VEL
LIN {X 0,Y 164.761,Z 267.955,A -85,B 0,C 180,E1 -23404.898,E2 -23404.898} C_VEL
LIN {X 0,Y 164.83,Z 267.938,A -85,B 0,C 180,E1 -23407.353,E2 -23407.353} C_VEL
LIN {X 0,Y 164.708,Z 267.967,A -85,B 0,C 180,E1 -23411.063,E2 -23411.063} C_VEL
LIN {X 0,Y 164.49,Z 267.987,A -85,B 0,C 180,E1 -23417.406,E2 -23417.406} C_VEL
LIN {X 0,Y 164.481,Z 267.996,A -85,B 0,C 180,E1 -23419.992,E2 -23419.992} C_VEL
LIN {X 0,Y 164.401,Z 268.006,A -85,B 0,C 180,E1 -23426.136,E2 -23426.136} C_VEL
LIN {X 0,Y 164.437,Z 268.076,A -85,B 0,C 180,E1 -23431.033,E2 -23431.033} C_VEL
LIN {X 0,Y 165.009,Z 271.738,A -85,B 0,C 180,E1 -23436.608,E2 -23436.608} C_VEL
LIN {X 0,Y 165.468,Z 274.191,A -85,B 0,C 180,E1 -23440.134,E2 -23440.134} C_VEL
LIN {X 0,Y 166.033,Z 276.967,A -85,B 0,C 180,E1 -23443.978,E2 -23443.978} C_VEL
LIN {X 0,Y 166.871,Z 281.071,A -85,B 0,C 180,E1 -23449.302,E2 -23449.302} C_VEL
LIN {X 0,Y 167.022,Z 282.75,A -85,B 0,C 180,E1 -23451.371,E2 -23451.371} C_VEL
LIN {X 0,Y 169.706,Z 296.405,A -85,B 0,C 180,E1 -23453.144,E2 -23453.144} C_VEL
LIN {X 0,Y 171.342,Z 309.43,A -85,B 0,C 180,E1 -23455.125,E2 -23455.125} C_VEL
LIN {X 0,Y 172.171,Z 321.755,A -85,B 0,C 180,E1 -23457.353,E2 -23457.353} C_VEL
LIN {X 0,Y 172.47,Z 332.726,A -85,B 0,C 180,E1 -23459.738,E2 -23459.738} C_VEL
LIN {X 0,Y 172.23,Z 343.96,A -85,B 0,C 180,E1 -23462.672,E2 -23462.672} C_VEL
LIN {X 0,Y 171.299,Z 348.051,A -85,B 0,C 180,E1 -23463.828,E2 -23463.828} C_VEL
LIN {X 0,Y 168.609,Z 357.493,A -85,B 0,C 180,E1 -23466.933,E2 -23466.933} C_VEL
LIN {X 0,Y 166.391,Z 365.459,A -85,B 0,C 180,E1 -23470.25,E2 -23470.25} C_VEL
LIN {X 0,Y 164.431,Z 372.311,A -85,B 0,C 180,E1 -23473.869,E2 -23473.869} C_VEL
LIN {X 0,Y 163.172,Z 377.803,A -85,B 0,C 180,E1 -23477.562,E2 -23477.562} C_VEL
LIN {X 0,Y 162.457,Z 382.08,A -85,B 0,C 180,E1 -23481.29,E2 -23481.29} C_VEL
LIN {X 0,Y 162.303,Z 385.264,A -85,B 0,C 180,E1 -23485.03,E2 -23485.03} C_VEL
LIN {X 0,Y 162.328,Z 386.81,A -85,B 0,C 180,E1 -23487.517,E2 -23487.517} C_VEL
LIN {X 0,Y 162.352,Z 387.928,A -85,B 0,C 180,E1 -23489.999,E2 -23489.999} C_VEL
LIN {X 0,Y 162.116,Z 388.819,A -85,B 0,C 180,E1 -23494.331,E2 -23494.331} C_VEL
LIN {X 0,Y 162.176,Z 388.694,A -85,B 0,C 180,E1 -23497.469,E2 -23497.469} C_VEL
LIN {X 0,Y 163.054,Z 387.311,A -85,B 0,C 180,E1 -23502.444,E2 -23502.444} C_VEL
LIN {X 0,Y 165.052,Z 384.34,A -85,B 0,C 180,E1 -23507.34,E2 -23507.34} C_VEL
LIN {X 0,Y 167.486,Z 381.093,A -85,B 0,C 180,E1 -23510.895,E2 -23510.895} C_VEL
LIN {X 0,Y 170.499,Z 376.867,A -85,B 0,C 180,E1 -23514.342,E2 -23514.342} C_VEL
LIN {X 0,Y 174.597,Z 370.567,A -85,B 0,C 180,E1 -23518.226,E2 -23518.226} C_VEL
LIN {X 0,Y 178.855,Z 363.965,A -85,B 0,C 180,E1 -23521.297,E2 -23521.297} C_VEL
LIN {X 0,Y 180.343,Z 360.633,A -85,B 0,C 180,E1 -23522.779,E2 -23522.779} C_VEL
LIN {X 0,Y 180.891,Z 357.381,A -85,B 0,C 180,E1 -23524.351,E2 -23524.351} C_VEL
LIN {X 0,Y 181.187,Z 348.337,A -85,B 0,C 180,E1 -23528.568,E2 -23528.568} C_VEL
LIN {X 0,Y 181.699,Z 345.766,A -85,B 0,C 180,E1 -23529.535,E2 -23529.535} C_VEL
LIN {X 0,Y 183.709,Z 337.146,A -85,B 0,C 180,E1 -23532.476,E2 -23532.476} C_VEL
LIN {X 0,Y 184.657,Z 329.478,A -85,B 0,C 180,E1 -23535.098,E2 -23535.098} C_VEL
LIN {X 0,Y 184.697,Z 326.355,A -85,B 0,C 180,E1 -23536.299,E2 -23536.299} C_VEL
LIN {X 0,Y 183.433,Z 320.22,A -85,B 0,C 180,E1 -23539.354,E2 -23539.354} C_VEL
LIN {X 0,Y 181.443,Z 313.27,A -85,B 0,C 180,E1 -23543.6,E2 -23543.6} C_VEL
LIN {X 0,Y 180.116,Z 308.85,A -85,B 0,C 180,E1 -23546.885,E2 -23546.885} C_VEL
LIN {X 0,Y 178.089,Z 302.279,A -85,B 0,C 180,E1 -23554.268,E2 -23554.268} C_VEL
LIN {X 0,Y 177.605,Z 300.769,A -85,B 0,C 180,E1 -23559.133,E2 -23559.133} C_VEL
LIN {X 0,Y 178.328,Z 300.372,A -85,B 0,C 180,E1 -23563.982,E2 -23563.982} C_VEL
LIN {X 0,Y 180.505,Z 303.847,A -85,B 0,C 180,E1 -23571.037,E2 -23571.037} C_VEL
LIN {X 0,Y 183.111,Z 308.83,A -85,B 0,C 180,E1 -23576.268,E2 -23576.268} C_VEL
LIN {X 0,Y 184.816,Z 314.167,A -85,B 0,C 180,E1 -23579.996,E2 -23579.996} C_VEL
LIN {X 0,Y 185.957,Z 318.673,A -85,B 0,C 180,E1 -23582.704,E2 -23582.704} C_VEL
LIN {X 0,Y 186.599,Z 324.583,A -85,B 0,C 180,E1 -23585.67,E2 -23585.67} C_VEL
LIN {X 0,Y 186.262,Z 331.598,A -85,B 0,C 180,E1 -23588.816,E2 -23588.816} C_VEL
LIN {X 0,Y 185.989,Z 333.861,A -85,B 0,C 180,E1 -23589.788,E2 -23589.788} C_VEL
LIN {X 0,Y 185.63,Z 334.859,A -85,B 0,C 180,E1 -23590.153,E2 -23590.153} C_VEL
LIN {X 0,Y 180.291,Z 343.752,A -85,B 0,C 180,E1 -23592.964,E2 -23592.964} C_VEL
LIN {X 0,Y 175.41,Z 350.963,A -85,B 0,C 180,E1 -23595.938,E2 -23595.938} C_VEL
LIN {X 0,Y 170.826,Z 357.029,A -85,B 0,C 180,E1 -23599.211,E2 -23599.211} C_VEL
LIN {X 0,Y 167.142,Z 361.455,A -85,B 0,C 180,E1 -23602.327,E2 -23602.327} C_VEL
LIN {X 0,Y 162.717,Z 366.168,A -85,B 0,C 180,E1 -23607.041,E2 -23607.041} C_VEL
LIN {X 0,Y 159.236,Z 369.203,A -85,B 0,C 180,E1 -23611.975,E2 -23611.975} C_VEL
LIN {X 0,Y 157.087,Z 370.491,A -85,B 0,C 180,E1 -23616.362,E2 -23616.362} C_VEL
LIN {X 0,Y 155.875,Z 370.702,A -85,B 0,C 180,E1 -23619.963,E2 -23619.963} C_VEL
LIN {X 0,Y 155.107,Z 370.125,A -85,B 0,C 180,E1 -23623.536,E2 -23623.536} C_VEL
LIN {X 0,Y 154.82,Z 368.836,A -85,B 0,C 180,E1 -23627.087,E2 -23627.087} C_VEL
LIN {X 0,Y 154.929,Z 366.864,A -85,B 0,C 180,E1 -23630.576,E2 -23630.576} C_VEL
LIN {X 0,Y 155.583,Z 363.8,A -85,B 0,C 180,E1 -23634.391,E2 -23634.391} C_VEL
